LIN {X 0,Y 202.13,Z 320.552,A -85,B 0,C 180,E1 -21800.081,E2 -21800.081} C_VEL
LIN {X 0,Y 203.145,Z 321.228,A -85,B 0,C 180,E1 -21800.929,E2 -21800.929} C_VEL
LIN {X 0,Y 205.158,Z 324.532,A -85,B 0,C 180,E1 -21802.673,E2 -21802.673} C_VEL
LIN {X 0,Y 207.742,Z 326.873,A -85,B 0,C 180,E1 -21804.538,E2 -21804.538} C_VEL
LIN {X 0,Y 210.085,Z 330.227,A -85,B 0,C 180,E1 -21806.178,E2 -21806.178} C_VEL
LIN {X 0,Y 211.841,Z 332.049,A -85,B 0,C 180,E1 -21807.274,E2 -21807.274} C_VEL
LIN {X 0,Y 214.755,Z 335.87,A -85,B 0,C 180,E1 -21809.025,E2 -21809.025} C_VEL
LIN {X 0,Y 219.434,Z 342.082,A -85,B 0,C 180,E1 -21811.565,E2 -21811.565} C_VEL
LIN {X 0,Y 223.531,Z 347.82,A -85,B 0,C 180,E1 -21813.584,E2 -21813.584} C_VEL
LIN {X 0,Y 230.012,Z 357.511,A -85,B 0,C 180,E1 -21816.473,E2 -21816.473} C_VEL
LIN {X 0,Y 236.957,Z 369.03,A -85,B 0,C 180,E1 -21819.257,E2 -21819.257} C_VEL
LIN {X 0,Y 243.804,Z 381.517,A -85,B 0,C 180,E1 -21821.753,E2 -21821.753} C_VEL
LIN {X 0,Y 244.17,Z 382.3,A -85,B 0,C 180,E1 -21821.884,E2 -21821.884} C_VEL
LIN {X 0,Y 239.074,Z 460.864,A -85,B 0,C 180,E1 -21824.002,E2 -21824.002} C_VEL
LIN {X 0,Y 237.145,Z 476.486,A -85,B 0,C 180,E1 -21824.661,E2 -21824.661} C_VEL
LIN {X 0,Y 234.514,Z 492.067,A -85,B 0,C 180,E1 -21825.681,E2 -21825.681} C_VEL
LIN {X 0,Y 231.128,Z 507.018,A -85,B 0,C 180,E1 -21827.007,E2 -21827.007} C_VEL
LIN {X 0,Y 227.337,Z 520.939,A -85,B 0,C 180,E1 -21828.638,E2 -21828.638} C_VEL
LIN {X 0,Y 222.831,Z 534.369,A -85,B 0,C 180,E1 -21830.598,E2 -21830.598} C_VEL
LIN {X 0,Y 218.143,Z 546.556,A -85,B 0,C 180,E1 -21832.836,E2 -21832.836} C_VEL
LIN {X 0,Y 213.369,Z 557.823,A -85,B 0,C 180,E1 -21835.433,E2 -21835.433} C_VEL
LIN {X 0,Y 209.266,Z 566.974,A -85,B 0,C 180,E1 -21838.064,E2 -21838.064} C_VEL
LIN {X 0,Y 204.762,Z 576.14,A -85,B 0,C 180,E1 -21841.28,E2 -21841.28} C_VEL
LIN {X 0,Y 201.404,Z 582.756,A -85,B 0,C 180,E1 -21844.138,E2 -21844.138} C_VEL
LIN {X 0,Y 197.654,Z 590.063,A -85,B 0,C 180,E1 -21848.077,E2 -21848.077} C_VEL
LIN {X 0,Y 194.772,Z 595.849,A -85,B 0,C 180,E1 -21852.138,E2 -21852.138} C_VEL
LIN {X 0,Y 193.112,Z 599.272,A -85,B 0,C 180,E1 -21855.24,E2 -21855.24} C_VEL
LIN {X 0,Y 191.574,Z 602.73,A -85,B 0,C 180,E1 -21859.429,E2 -21859.429} C_VEL
LIN {X 0,Y 190.735,Z 605.008,A -85,B 0,C 180,E1 -21863.652,E2 -21863.652} C_VEL
LIN {X 0,Y 190.443,Z 606.165,A -85,B 0,C 180,E1 -21867.884,E2 -21867.884} C_VEL
LIN {X 0,Y 190.442,Z 606.176,A -85,B 0,C 180,E1 -21872.114,E2 -21872.114} C_VEL
LIN {X 0,Y 190.734,Z 605.068,A -85,B 0,C 180,E1 -21876.346,E2 -21876.346} C_VEL
LIN {X 0,Y 191.569,Z 602.836,A -85,B 0,C 180,E1 -21880.569,E2 -21880.569} C_VEL
LIN {X 0,Y 193.074,Z 599.42,A -85,B 0,C 180,E1 -21884.761,E2 -21884.761} C_VEL
LIN {X 0,Y 195.42,Z 594.732,A -85,B 0,C 180,E1 -21888.884,E2 -21888.884} C_VEL
LIN {X 0,Y 198.471,Z 588.575,A -85,B 0,C 180,E1 -21892.974,E2 -21892.974} C_VEL
LIN {X 0,Y 202.417,Z 580.99,A -85,B 0,C 180,E1 -21896.83,E2 -21896.83} C_VEL
LIN {X 0,Y 206.506,Z 572.813,A -85,B 0,C 180,E1 -21900.13,E2 -21900.13} C_VEL
LIN {X 0,Y 211.148,Z 563.18,A -85,B 0,C 180,E1 -21903.226,E2 -21903.226} C_VEL
LIN {X 0,Y 215.623,Z 552.84,A -85,B 0,C 180,E1 -21905.921,E2 -21905.921} C_VEL
LIN {X 0,Y 220.595,Z 540.782,A -85,B 0,C 180,E1 -21908.407,E2 -21908.407} C_VEL
LIN {X 0,Y 224.945,Z 528.686,A -85,B 0,C 180,E1 -21910.412,E2 -21910.412} C_VEL
LIN {X 0,Y 228.967,Z 515.537,A -85,B 0,C 180,E1 -21912.177,E2 -21912.177} C_VEL
LIN {X 0,Y 232.029,Z 503.75,A -85,B 0,C 180,E1 -21913.442,E2 -21913.442} C_VEL
LIN {X 0,Y 235.137,Z 489.584,A -85,B 0,C 180,E1 -21914.618,E2 -21914.618} C_VEL
LIN {X 0,Y 237.476,Z 475.706,A -85,B 0,C 180,E1 -21915.482,E2 -21915.482} C_VEL
LIN {X 0,Y 239.05,Z 462.425,A -85,B 0,C 180,E1 -21916.078,E2 -21916.078} C_VEL
LIN {X 0,Y 243.886,Z 390.726,A -85,B 0,C 180,E1 -21917.99,E2 -21917.99} C_VEL
LIN {X 0,Y 244.24,Z 382.256,A -85,B 0,C 180,E1 -21918.264,E2 -21918.264} C_VEL
LIN {X 0,Y 237.424,Z 369.67,A -85,B 0,C 180,E1 -21920.748,E2 -21920.748} C_VEL
LIN {X 0,Y 230.601,Z 358.379,A -85,B 0,C 180,E1 -21923.469,E2 -21923.469} C_VEL
LIN {X 0,Y 224.172,Z 348.632,A -85,B 0,C 180,E1 -21926.322,E2 -21926.322} C_VEL
LIN {X 0,Y 218.479,Z 340.65,A -85,B 0,C 180,E1 -21929.158,E2 -21929.158} C_VEL
LIN {X 0,Y 214.78,Z 335.855,A -85,B 0,C 180,E1 -21931.197,E2 -21931.197} C_VEL
LIN {X 0,Y 211.989,Z 332.222,A -85,B 0,C 180,E1 -21932.88,E2 -21932.88} C_VEL
LIN {X 0,Y 210.588,Z 330.732,A -85,B 0,C 180,E1 -21933.756,E2 -21933.756} C_VEL
LIN {X 0,Y 207.985,Z 327.314,A -85,B 0,C 180,E1 -21935.547,E2 -21935.547} C_VEL
LIN {X 0,Y 207.379,Z 326.351,A -85,B 0,C 180,E1 -21936.004,E2 -21936.004} C_VEL
LIN {X 0,Y 204.867,Z 324.176,A -85,B 0,C 180,E1 -21937.854,E2 -21937.854} C_VEL
LIN {X 0,Y 203.045,Z 321.01,A -85,B 0,C 180,E1 -21939.485,E2 -21939.485} C_VEL
LIN {X 0,Y 200.267,Z 319.057,A -85,B 0,C 180,E1 -21941.983,E2 -21941.983} C_VEL
LIN {X 0,Y 198.467,Z 316.064,A -85,B 0,C 180,E1 -21944.071,E2 -21944.071} C_VEL
LIN {X 0,Y 198.111,Z 315.123,A -85,B 0,C 180,E1 -21944.57,E2 -21944.57} C_VEL
LIN {X 0,Y 195.257,Z 313.598,A -85,B 0,C 180,E1 -21948.319,E2 -21948.319} C_VEL
LIN {X 0,Y 193.137,Z 309.963,A -85,B 0,C 180,E1 -21953.077,E2 -21953.077} C_VEL
LIN {X 0,Y 192.954,Z 309.07,A -85,B 0,C 180,E1 -21953.989,E2 -21953.989} C_VEL
LIN {X 0,Y 193.233,Z 309.035,A -85,B 0,C 180,E1 -21957.915,E2 -21957.915} C_VEL
LIN {X 0,Y 193.412,Z 309.003,A -85,B 0,C 180,E1 -21960,E2 -21960} C_VEL
LIN {X 0,Y 192.951,Z 309.06,A -85,B 0,C 180,E1 -21965.224,E2 -21965.224} C_VEL
LIN {X 0,Y 193,Z 309.378,A -85,B 0,C 180,E1 -21965.878,E2 -21965.878} C_VEL
LIN {X 0,Y 194.263,Z 312.349,A -85,B 0,C 180,E1 -21969.369,E2 -21969.369} C_VEL
LIN {X 0,Y 196.824,Z 314.644,A -85,B 0,C 180,E1 -21973.42,E2 -21973.42} C_VEL
LIN {X 0,Y 198.338,Z 315.385,A -85,B 0,C 180,E1 -21975.214,E2 -21975.214} C_VEL
LIN {X 0,Y 199.492,Z 317.921,A -85,B 0,C 180,E1 -21976.681,E2 -21976.681} C_VEL
LIN {X 0,Y 201.693,Z 320.181,A -85,B 0,C 180,E1 -21978.869,E2 -21978.869} C_VEL
LIN {X 0,Y 203.142,Z 321.115,A -85,B 0,C 180,E1 -21980.109,E2 -21980.109} C_VEL
LIN {X 0,Y 204.86,Z 324.08,A -85,B 0,C 180,E1 -21981.641,E2 -21981.641} C_VEL
LIN {X 0,Y 207.774,Z 326.812,A -85,B 0,C 180,E1 -21983.79,E2 -21983.79} C_VEL
LIN {X 0,Y 210.353,Z 330.409,A -85,B 0,C 180,E1 -21985.597,E2 -21985.597} C_VEL
LIN {X 0,Y 211.92,Z 332.086,A -85,B 0,C 180,E1 -21986.582,E2 -21986.582} C_VEL
LIN {X 0,Y 214.986,Z 336.068,A -85,B 0,C 180,E1 -21988.428,E2 -21988.428} C_VEL
LIN {X 0,Y 219.53,Z 343.033,A -85,B 0,C 180,E1 -21990.96,E2 -21990.96} C_VEL
LIN {X 0,Y 223.296,Z 349.285,A -85,B 0,C 180,E1 -21992.883,E2 -21992.883} C_VEL
LIN {X 0,Y 227.557,Z 356.613,A -85,B 0,C 180,E1 -21994.888,E2 -21994.888} C_VEL
LIN {X 0,Y 228.819,Z 359.483,A -85,B 0,C 180,E1 -21995.486,E2 -21995.486} C_VEL
LIN {X 0,Y 230.208,Z 364.449,A -85,B 0,C 180,E1 -21996.22,E2 -21996.22} C_VEL
LIN {X 0,Y 233.07,Z 378.716,A -85,B 0,C 180,E1 -21997.864,E2 -21997.864} C_VEL
LIN {X 0,Y 234.805,Z 383.494,A -85,B 0,C 180,E1 -21998.63,E2 -21998.63} C_VEL
LIN {X 0,Y 238.967,Z 393.731,A -85,B 0,C 180,E1 -22000.317,E2 -22000.317} C_VEL
LIN {X 0,Y 235.291,Z 450.409,A -85,B 0,C 180,E1 -22001.853,E2 -22001.853} C_VEL
LIN {X 0,Y 233.436,Z 475.234,A -85,B 0,C 180,E1 -22002.552,E2 -22002.552} C_VEL
LIN {X 0,Y 231.252,Z 490.946,A -85,B 0,C 180,E1 -22003.245,E2 -22003.245} C_VEL
LIN {X 0,Y 228.371,Z 505.434,A -85,B 0,C 180,E1 -22004.158,E2 -22004.158} C_VEL
LIN {X 0,Y 224.872,Z 519.174,A -85,B 0,C 180,E1 -22005.317,E2 -22005.317} C_VEL
LIN {X 0,Y 220.787,Z 532.642,A -85,B 0,C 180,E1 -22006.814,E2 -22006.814} C_VEL
LIN {X 0,Y 216.512,Z 544.93,A -85,B 0,C 180,E1 -22008.562,E2 -22008.562} C_VEL
LIN {X 0,Y 211.366,Z 557.724,A -85,B 0,C 180,E1 -22010.821,E2 -22010.821} C_VEL
LIN {X 0,Y 206.254,Z 569.229,A -85,B 0,C 180,E1 -22013.395,E2 -22013.395} C_VEL
LIN {X 0,Y 201.601,Z 578.92,A -85,B 0,C 180,E1 -22016.099,E2 -22016.099} C_VEL
LIN {X 0,Y 196.862,Z 588.577,A -85,B 0,C 180,E1 -22019.481,E2 -22019.481} C_VEL
LIN {X 0,Y 192.876,Z 596.405,A -85,B 0,C 180,E1 -22022.906,E2 -22022.906} C_VEL
LIN {X 0,Y 189.093,Z 603.84,A -85,B 0,C 180,E1 -22027.031,E2 -22027.031} C_VEL
LIN {X 0,Y 186.295,Z 609.751,A -85,B 0,C 180,E1 -22031.298,E2 -22031.298} C_VEL
LIN {X 0,Y 184.799,Z 613.274,A -85,B 0,C 180,E1 -22034.562,E2 -22034.562} C_VEL
LIN {X 0,Y 183.53,Z 616.842,A -85,B 0,C 180,E1 -22038.963,E2 -22038.963} C_VEL
LIN {X 0,Y 183.109,Z 619.202,A -85,B 0,C 180,E1 -22043.389,E2 -22043.389} C_VEL
LIN {X 0,Y 183.13,Z 620.394,A -85,B 0,C 180,E1 -22047.802,E2 -22047.802} C_VEL
LIN {X 0,Y 183.283,Z 620.556,A -85,B 0,C 180,E1 -22050.001,E2 -22050.001} C_VEL
LIN {X 0,Y 183.114,Z 619.928,A -85,B 0,C 180,E1 -22054.403,E2 -22054.403} C_VEL
LIN {X 0,Y 183.241,Z 618.133,A -85,B 0,C 180,E1 -22058.826,E2 -22058.826} C_VEL
LIN {X 0,Y 184.022,Z 615.159,A -85,B 0,C 180,E1 -22063.248,E2 -22063.248} C_VEL
LIN {X 0,Y 185.723,Z 610.945,A -85,B 0,C 180,E1 -22067.623,E2 -22067.623} C_VEL
LIN {X 0,Y 188.26,Z 605.378,A -85,B 0,C 180,E1 -22071.921,E2 -22071.921} C_VEL
LIN {X 0,Y 191.758,Z 598.315,A -85,B 0,C 180,E1 -22076.093,E2 -22076.093} C_VEL
LIN {X 0,Y 195.731,Z 590.779,A -85,B 0,C 180,E1 -22079.586,E2 -22079.586} C_VEL
LIN {X 0,Y 200.221,Z 581.697,A -85,B 0,C 180,E1 -22082.962,E2 -22082.962} C_VEL
LIN {X 0,Y 205.441,Z 570.793,A -85,B 0,C 180,E1 -22086.166,E2 -22086.166} C_VEL
LIN {X 0,Y 210.422,Z 559.576,A -85,B 0,C 180,E1 -22088.775,E2 -22088.775} C_VEL
LIN {X 0,Y 215.782,Z 546.661,A -85,B 0,C 180,E1 -22091.121,E2 -22091.121} C_VEL
LIN {X 0,Y 220.293,Z 533.792,A -85,B 0,C 180,E1 -22092.996,E2 -22092.996} C_VEL
LIN {X 0,Y 224.342,Z 520.525,A -85,B 0,C 180,E1 -22094.504,E2 -22094.504} C_VEL
LIN {X 0,Y 227.806,Z 507.143,A -85,B 0,C 180,E1 -22095.673,E2 -22095.673} C_VEL
LIN {X 0,Y 230.83,Z 492.493,A -85,B 0,C 180,E1 -22096.63,E2 -22096.63} C_VEL
LIN {X 0,Y 232.989,Z 477.524,A -85,B 0,C 180,E1 -22097.331,E2 -22097.331} C_VEL
LIN {X 0,Y 234.684,Z 457.569,A -85,B 0,C 180,E1 -22097.913,E2 -22097.913} C_VEL
LIN {X 0,Y 238.816,Z 393.594,A -85,B 0,C 180,E1 -22099.652,E2 -22099.652} C_VEL
LIN {X 0,Y 233.193,Z 380.016,A -85,B 0,C 180,E1 -22101.945,E2 -22101.945} C_VEL
LIN {X 0,Y 227.753,Z 368.646,A -85,B 0,C 180,E1 -22104.303,E2 -22104.303} C_VEL
LIN {X 0,Y 221.581,Z 356.972,A -85,B 0,C 180,E1 -22107.236,E2 -22107.236} C_VEL
LIN {X 0,Y 215.921,Z 347.368,A -85,B 0,C 180,E1 -22110.24,E2 -22110.24} C_VEL
LIN {X 0,Y 212.629,Z 342.242,A -85,B 0,C 180,E1 -22112.169,E2 -22112.169} C_VEL
LIN {X 0,Y 208.968,Z 337.475,A -85,B 0,C 180,E1 -22114.475,E2 -22114.475} C_VEL
LIN {X 0,Y 206.188,Z 333.97,A -85,B 0,C 180,E1 -22116.414,E2 -22116.414} C_VEL
LIN {X 0,Y 205.461,Z 332.88,A -85,B 0,C 180,E1 -22116.971,E2 -22116.971} C_VEL
LIN {X 0,Y 202.738,Z 330.139,A -85,B 0,C 180,E1 -22119.088,E2 -22119.088} C_VEL
LIN {X 0,Y 201.362,Z 327.685,A -85,B 0,C 180,E1 -22120.371,E2 -22120.371} C_VEL
LIN {X 0,Y 198.647,Z 325.483,A -85,B 0,C 180,E1 -22122.918,E2 -22122.918} C_VEL
LIN {X 0,Y 196.975,Z 322.515,A -85,B 0,C 180,E1 -22124.942,E2 -22124.942} C_VEL
LIN {X 0,Y 196.531,Z 321.931,A -85,B 0,C 180,E1 -22125.504,E2 -22125.504} C_VEL
LIN {X 0,Y 193.771,Z 320.059,A -85,B 0,C 180,E1 -22129.354,E2 -22129.354} C_VEL
LIN {X 0,Y 192.084,Z 316.757,A -85,B 0,C 180,E1 -22133.303,E2 -22133.303} C_VEL
LIN {X 0,Y 191.818,Z 316.073,A -85,B 0,C 180,E1 -22134.217,E2 -22134.217} C_VEL
LIN {X 0,Y 190.8,Z 315.614,A -85,B 0,C 180,E1 -22140,E2 -22140} C_VEL
LIN {X 0,Y 192.014,Z 316.301,A -85,B 0,C 180,E1 -22146.964,E2 -22146.964} C_VEL
LIN {X 0,Y 193.236,Z 319.399,A -85,B 0,C 180,E1 -22150.234,E2 -22150.234} C_VEL
LIN {X 0,Y 195.466,Z 321.51,A -85,B 0,C 180,E1 -22153.781,E2 -22153.781} C_VEL
LIN {X 0,Y 196.819,Z 322.191,A -85,B 0,C 180,E1 -22155.428,E2 -22155.428} C_VEL
LIN {X 0,Y 198.612,Z 325.558,A -85,B 0,C 180,E1 -22157.64,E2 -22157.64} C_VEL
LIN {X 0,Y 201.56,Z 328.097,A -85,B 0,C 180,E1 -22160.407,E2 -22160.407} C_VEL
LIN {X 0,Y 203.71,Z 331.392,A -85,B 0,C 180,E1 -22162.303,E2 -22162.303} C_VEL
LIN {X 0,Y 205.811,Z 333.361,A -85,B 0,C 180,E1 -22163.876,E2 -22163.876} C_VEL
LIN {X 0,Y 208.392,Z 336.945,A -85,B 0,C 180,E1 -22165.735,E2 -22165.735} C_VEL
LIN {X 0,Y 209.758,Z 338.468,A -85,B 0,C 180,E1 -22166.624,E2 -22166.624} C_VEL
LIN {X 0,Y 212.93,Z 342.541,A -85,B 0,C 180,E1 -22168.584,E2 -22168.584} C_VEL
LIN {X 0,Y 219.429,Z 351.601,A -85,B 0,C 180,E1 -22172.146,E2 -22172.146} C_VEL
LIN {X 0,Y 226.743,Z 362.814,A -85,B 0,C 180,E1 -22175.613,E2 -22175.613} C_VEL
LIN {X 0,Y 233.269,Z 373.858,A -85,B 0,C 180,E1 -22178.36,E2 -22178.36} C_VEL
LIN {X 0,Y 239.321,Z 385.095,A -85,B 0,C 180,E1 -22180.686,E2 -22180.686} C_VEL
LIN {X 0,Y 234.217,Z 461.153,A -85,B 0,C 180,E1 -22182.757,E2 -22182.757} C_VEL
LIN {X 0,Y 232.232,Z 476.767,A -85,B 0,C 180,E1 -22183.421,E2 -22183.421} C_VEL
LIN {X 0,Y 229.486,Z 492.346,A -85,B 0,C 180,E1 -22184.442,E2 -22184.442} C_VEL
LIN {X 0,Y 226.006,Z 507.293,A -85,B 0,C 180,E1 -22185.785,E2 -22185.785} C_VEL
LIN {X 0,Y 222.066,Z 521.214,A -85,B 0,C 180,E1 -22187.429,E2 -22187.429} C_VEL
LIN {X 0,Y 217.393,Z 534.643,A -85,B 0,C 180,E1 -22189.411,E2 -22189.411} C_VEL
LIN {X 0,Y 212.518,Z 546.83,A -85,B 0,C 180,E1 -22191.678,E2 -22191.678} C_VEL
LIN {X 0,Y 207.556,Z 558.097,A -85,B 0,C 180,E1 -22194.32,E2 -22194.32} C_VEL
LIN {X 0,Y 202.524,Z 568.691,A -85,B 0,C 180,E1 -22197.459,E2 -22197.459} C_VEL
LIN {X 0,Y 197.926,Z 577.626,A -85,B 0,C 180,E1 -22200.774,E2 -22200.774} C_VEL
LIN {X 0,Y 193.952,Z 585.023,A -85,B 0,C 180,E1 -22204.224,E2 -22204.224} C_VEL
LIN {X 0,Y 190.243,Z 591.928,A -85,B 0,C 180,E1 -22208.319,E2 -22208.319} C_VEL
LIN {X 0,Y 187.299,Z 597.347,A -85,B 0,C 180,E1 -22212.53,E2 -22212.53} C_VEL
LIN {X 0,Y 185.313,Z 601.425,A -85,B 0,C 180,E1 -22216.846,E2 -22216.846} C_VEL
LIN {X 0,Y 184.05,Z 604.284,A -85,B 0,C 180,E1 -22221.213,E2 -22221.213} C_VEL
LIN {X 0,Y 183.449,Z 605.995,A -85,B 0,C 180,E1 -22225.605,E2 -22225.605} C_VEL
LIN {X 0,Y 183.336,Z 606.589,A -85,B 0,C 180,E1 -22229.999,E2 -22229.999} C_VEL
LIN {X 0,Y 183.449,Z 606.031,A -85,B 0,C 180,E1 -22234.393,E2 -22234.393} C_VEL
LIN {X 0,Y 184.048,Z 604.366,A -85,B 0,C 180,E1 -22238.785,E2 -22238.785} C_VEL
LIN {X 0,Y 185.295,Z 601.551,A -85,B 0,C 180,E1 -22243.153,E2 -22243.153} C_VEL
LIN {X 0,Y 187.249,Z 597.515,A -85,B 0,C 180,E1 -22247.472,E2 -22247.472} C_VEL
LIN {X 0,Y 190.147,Z 592.15,A -85,B 0,C 180,E1 -22251.69,E2 -22251.69} C_VEL
LIN {X 0,Y 193.855,Z 585.308,A -85,B 0,C 180,E1 -22255.787,E2 -22255.787} C_VEL
LIN {X 0,Y 198.454,Z 576.755,A -85,B 0,C 180,E1 -22259.721,E2 -22259.721} C_VEL
LIN {X 0,Y 203.204,Z 567.65,A -85,B 0,C 180,E1 -22263.005,E2 -22263.005} C_VEL
LIN {X 0,Y 207.421,Z 558.546,A -85,B 0,C 180,E1 -22265.705,E2 -22265.705} C_VEL
LIN {X 0,Y 212.458,Z 547.353,A -85,B 0,C 180,E1 -22268.333,E2 -22268.333} C_VEL
LIN {X 0,Y 217.255,Z 535.27,A -85,B 0,C 180,E1 -22270.618,E2 -22270.618} C_VEL
LIN {X 0,Y 221.912,Z 521.99,A -85,B 0,C 180,E1 -22272.605,E2 -22272.605} C_VEL
LIN {X 0,Y 225.604,Z 509.172,A -85,B 0,C 180,E1 -22274.151,E2 -22274.151} C_VEL
LIN {X 0,Y 229.127,Z 494.706,A -85,B 0,C 180,E1 -22275.49,E2 -22275.49} C_VEL
LIN {X 0,Y 231.901,Z 480.025,A -85,B 0,C 180,E1 -22276.505,E2 -22276.505} C_VEL
LIN {X 0,Y 233.94,Z 464.955,A -85,B 0,C 180,E1 -22277.234,E2 -22277.234} C_VEL
LIN {X 0,Y 235.343,Z 448.353,A -85,B 0,C 180,E1 -22277.734,E2 -22277.734} C_VEL
LIN {X 0,Y 239.471,Z 385.303,A -85,B 0,C 180,E1 -22279.433,E2 -22279.433} C_VEL
LIN {X 0,Y 232.955,Z 373.112,A -85,B 0,C 180,E1 -22281.956,E2 -22281.956} C_VEL
LIN {X 0,Y 226.004,Z 361.512,A -85,B 0,C 180,E1 -22284.917,E2 -22284.917} C_VEL
LIN {X 0,Y 218.751,Z 350.547,A -85,B 0,C 180,E1 -22288.42,E2 -22288.42} C_VEL
LIN {X 0,Y 214.628,Z 345.033,A -85,B 0,C 180,E1 -22290.647,E2 -22290.647} C_VEL
LIN {X 0,Y 212.452,Z 342.032,A -85,B 0,C 180,E1 -22291.931,E2 -22291.931} C_VEL
LIN {X 0,Y 209.066,Z 337.592,A -85,B 0,C 180,E1 -22294.086,E2 -22294.086} C_VEL
LIN {X 0,Y 206.32,Z 334.216,A -85,B 0,C 180,E1 -22296.006,E2 -22296.006} C_VEL
LIN {X 0,Y 205.42,Z 332.907,A -85,B 0,C 180,E1 -22296.697,E2 -22296.697} C_VEL
LIN {X 0,Y 202.711,Z 330.117,A -85,B 0,C 180,E1 -22298.838,E2 -22298.838} C_VEL
LIN {X 0,Y 201.303,Z 327.686,A -85,B 0,C 180,E1 -22300.165,E2 -22300.165} C_VEL
LIN {X 0,Y 198.685,Z 325.586,A -85,B 0,C 180,E1 -22302.661,E2 -22302.661} C_VEL
LIN {X 0,Y 196.905,Z 322.419,A -85,B 0,C 180,E1 -22304.87,E2 -22304.87} C_VEL
LIN {X 0,Y 196.412,Z 321.915,A -85,B 0,C 180,E1 -22305.494,E2 -22305.494} C_VEL
LIN {X 0,Y 193.762,Z 320.069,A -85,B 0,C 180,E1 -22309.367,E2 -22309.367} C_VEL
LIN {X 0,Y 191.99,Z 316.273,A -85,B 0,C 180,E1 -22314.09,E2 -22314.09} C_VEL
LIN {X 0,Y 191.122,Z 315.724,A -85,B 0,C 180,E1 -22320,E2 -22320} C_VEL
LIN {X 0,Y 191.984,Z 316.219,A -85,B 0,C 180,E1 -22325.382,E2 -22325.382} C_VEL
LIN {X 0,Y 193.28,Z 319.362,A -85,B 0,C 180,E1 -22329.175,E2 -22329.175} C_VEL
LIN {X 0,Y 195.593,Z 321.528,A -85,B 0,C 180,E1 -22332.978,E2 -22332.978} C_VEL
LIN {X 0,Y 196.899,Z 322.186,A -85,B 0,C 180,E1 -22334.601,E2 -22334.601} C_VEL
LIN {X 0,Y 198.354,Z 325.041,A -85,B 0,C 180,E1 -22336.466,E2 -22336.466} C_VEL
LIN {X 0,Y 200.658,Z 327.228,A -85,B 0,C 180,E1 -22338.771,E2 -22338.771} C_VEL
LIN {X 0,Y 201.545,Z 327.96,A -85,B 0,C 180,E1 -22339.564,E2 -22339.564} C_VEL
LIN {X 0,Y 203.71,Z 331.292,A -85,B 0,C 180,E1 -22341.504,E2 -22341.504} C_VEL
LIN {X 0,Y 205.872,Z 333.311,A -85,B 0,C 180,E1 -22343.14,E2 -22343.14} C_VEL
LIN {X 0,Y 208.65,Z 337.112,A -85,B 0,C 180,E1 -22345.146,E2 -22345.146} C_VEL
LIN {X 0,Y 210.023,Z 338.805,A -85,B 0,C 180,E1 -22346.053,E2 -22346.053} C_VEL
LIN {X 0,Y 213.649,Z 343.667,A -85,B 0,C 180,E1 -22348.294,E2 -22348.294} C_VEL
LIN {X 0,Y 217.814,Z 350.47,A -85,B 0,C 180,E1 -22350.677,E2 -22350.677} C_VEL
LIN {X 0,Y 222.059,Z 357.794,A -85,B 0,C 180,E1 -22352.887,E2 -22352.887} C_VEL
LIN {X 0,Y 227.28,Z 367.659,A -85,B 0,C 180,E1 -22355.38,E2 -22355.38} C_VEL
LIN {X 0,Y 232.625,Z 378.602,A -85,B 0,C 180,E1 -22357.719,E2 -22357.719} C_VEL
LIN {X 0,Y 234.805,Z 383.494,A -85,B 0,C 180,E1 -22358.63,E2 -22358.63} C_VEL
LIN {X 0,Y 235.574,Z 386.228,A -85,B 0,C 180,E1 -22358.99,E2 -22358.99} C_VEL
LIN {X 0,Y 235.666,Z 390.703,A -85,B 0,C 180,E1 -22359.228,E2 -22359.228} C_VEL
LIN {X 0,Y 233.874,Z 403.174,A -85,B 0,C 180,E1 -22359.285,E2 -22359.285} C_VEL
LIN {X 0,Y 233.774,Z 404.58,A -85,B 0,C 180,E1 -22359.322,E2 -22359.322} C_VEL
LIN {X 0,Y 228.83,Z 473.789,A -85,B 0,C 180,E1 -22361.197,E2 -22361.197} C_VEL
LIN {X 0,Y 226.566,Z 489.92,A -85,B 0,C 180,E1 -22361.887,E2 -22361.887} C_VEL
LIN {X 0,Y 223.458,Z 505.169,A -85,B 0,C 180,E1 -22362.846,E2 -22362.846} C_VEL
LIN {X 0,Y 219.862,Z 518.908,A -85,B 0,C 180,E1 -22364.011,E2 -22364.011} C_VEL
LIN {X 0,Y 215.646,Z 532.376,A -85,B 0,C 180,E1 -22365.518,E2 -22365.518} C_VEL
LIN {X 0,Y 211.045,Z 545.121,A -85,B 0,C 180,E1 -22367.353,E2 -22367.353} C_VEL
LIN {X 0,Y 205.879,Z 557.456,A -85,B 0,C 180,E1 -22369.565,E2 -22369.565} C_VEL
LIN {X 0,Y 200.564,Z 568.959,A -85,B 0,C 180,E1 -22372.178,E2 -22372.178} C_VEL
LIN {X 0,Y 195.692,Z 578.649,A -85,B 0,C 180,E1 -22374.928,E2 -22374.928} C_VEL
LIN {X 0,Y 190.911,Z 587.945,A -85,B 0,C 180,E1 -22378.242,E2 -22378.242} C_VEL
LIN {X 0,Y 186.513,Z 596.133,A -85,B 0,C 180,E1 -22381.901,E2 -22381.901} C_VEL
LIN {X 0,Y 182.497,Z 603.567,A -85,B 0,C 180,E1 -22386.15,E2 -22386.15} C_VEL
LIN {X 0,Y 179.513,Z 609.478,A -85,B 0,C 180,E1 -22390.564,E2 -22390.564} C_VEL
LIN {X 0,Y 177.901,Z 613.002,A -85,B 0,C 180,E1 -22393.948,E2 -22393.948} C_VEL
LIN {X 0,Y 176.508,Z 616.57,A -85,B 0,C 180,E1 -22398.518,E2 -22398.518} C_VEL
LIN {X 0,Y 176.013,Z 618.93,A -85,B 0,C 180,E1 -22403.121,E2 -22403.121} C_VEL
LIN {X 0,Y 176.015,Z 619.921,A -85,B 0,C 180,E1 -22406.569,E2 -22406.569} C_VEL
LIN {X 0,Y 176.185,Z 620.285,A -85,B 0,C 180,E1 -22410.001,E2 -22410.001} C_VEL
LIN {X 0,Y 176.019,Z 619.657,A -85,B 0,C 180,E1 -22414.581,E2 -22414.581} C_VEL
LIN {X 0,Y 176.19,Z 617.861,A -85,B 0,C 180,E1 -22419.182,E2 -22419.182} C_VEL
LIN {X 0,Y 177.051,Z 614.885,A -85,B 0,C 180,E1 -22423.78,E2 -22423.78} C_VEL
LIN {X 0,Y 178.906,Z 610.671,A -85,B 0,C 180,E1 -22428.318,E2 -22428.318} C_VEL
LIN {X 0,Y 181.61,Z 605.103,A -85,B 0,C 180,E1 -22432.768,E2 -22432.768} C_VEL
LIN {X 0,Y 185.338,Z 598.04,A -85,B 0,C 180,E1 -22437.069,E2 -22437.069} C_VEL
LIN {X 0,Y 189.49,Z 590.503,A -85,B 0,C 180,E1 -22440.663,E2 -22440.663} C_VEL
LIN {X 0,Y 194.241,Z 581.421,A -85,B 0,C 180,E1 -22444.114,E2 -22444.114} C_VEL
LIN {X 0,Y 199.712,Z 570.518,A -85,B 0,C 180,E1 -22447.377,E2 -22447.377} C_VEL
LIN {X 0,Y 204.919,Z 559.302,A -85,B 0,C 180,E1 -22450.022,E2 -22450.022} C_VEL
LIN {X 0,Y 210.373,Z 546.589,A -85,B 0,C 180,E1 -22452.366,E2 -22452.366} C_VEL
LIN {X 0,Y 215.14,Z 533.516,A -85,B 0,C 180,E1 -22454.289,E2 -22454.289} C_VEL
LIN {X 0,Y 219.305,Z 520.248,A -85,B 0,C 180,E1 -22455.813,E2 -22455.813} C_VEL
LIN {X 0,Y 222.878,Z 506.864,A -85,B 0,C 180,E1 -22456.986,E2 -22456.986} C_VEL
LIN {X 0,Y 226.014,Z 492.213,A -85,B 0,C 180,E1 -22457.938,E2 -22457.938} C_VEL
LIN {X 0,Y 228.247,Z 477.24,A -85,B 0,C 180,E1 -22458.638,E2 -22458.638} C_VEL
LIN {X 0,Y 229.989,Z 457.277,A -85,B 0,C 180,E1 -22459.225,E2 -22459.225} C_VEL
LIN {X 0,Y 234.146,Z 396.149,A -85,B 0,C 180,E1 -22460.881,E2 -22460.881} C_VEL
LIN {X 0,Y 228.792,Z 383.138,A -85,B 0,C 180,E1 -22463.201,E2 -22463.201} C_VEL
LIN {X 0,Y 223.37,Z 371.735,A -85,B 0,C 180,E1 -22465.709,E2 -22465.709} C_VEL
LIN {X 0,Y 218.249,Z 361.872,A -85,B 0,C 180,E1 -22468.306,E2 -22468.306} C_VEL
LIN {X 0,Y 213.174,Z 352.979,A -85,B 0,C 180,E1 -22471.159,E2 -22471.159} C_VEL
LIN {X 0,Y 210.264,Z 348.333,A -85,B 0,C 180,E1 -22472.952,E2 -22472.952} C_VEL
LIN {X 0,Y 206.729,Z 343.627,A -85,B 0,C 180,E1 -22475.289,E2 -22475.289} C_VEL
LIN {X 0,Y 203.919,Z 339.743,A -85,B 0,C 180,E1 -22477.381,E2 -22477.381} C_VEL
LIN {X 0,Y 200.753,Z 336.231,A -85,B 0,C 180,E1 -22479.976,E2 -22479.976} C_VEL
LIN {X 0,Y 199.706,Z 334.347,A -85,B 0,C 180,E1 -22481.003,E2 -22481.003} C_VEL
LIN {X 0,Y 197.123,Z 332.045,A -85,B 0,C 180,E1 -22483.561,E2 -22483.561} C_VEL
LIN {X 0,Y 195.266,Z 328.846,A -85,B 0,C 180,E1 -22485.94,E2 -22485.94} C_VEL
LIN {X 0,Y 192.666,Z 326.943,A -85,B 0,C 180,E1 -22489.735,E2 -22489.735} C_VEL
LIN {X 0,Y 191.011,Z 323.457,A -85,B 0,C 180,E1 -22493.928,E2 -22493.928} C_VEL
LIN {X 0,Y 190.784,Z 323.072,A -85,B 0,C 180,E1 -22494.716,E2 -22494.716} C_VEL
LIN {X 0,Y 190.016,Z 322.767,A -85,B 0,C 180,E1 -22502.12,E2 -22502.12} C_VEL
LIN {X 0,Y 191.031,Z 323.349,A -85,B 0,C 180,E1 -22506.671,E2 -22506.671} C_VEL
LIN {X 0,Y 192.218,Z 326.384,A -85,B 0,C 180,E1 -22509.982,E2 -22509.982} C_VEL
LIN {X 0,Y 194.429,Z 328.503,A -85,B 0,C 180,E1 -22513.589,E2 -22513.589} C_VEL
LIN {X 0,Y 195.512,Z 329.22,A -85,B 0,C 180,E1 -22514.973,E2 -22514.973} C_VEL
LIN {X 0,Y 197.475,Z 332.617,A -85,B 0,C 180,E1 -22517.425,E2 -22517.425} C_VEL
LIN {X 0,Y 199.963,Z 334.84,A -85,B 0,C 180,E1 -22519.84,E2 -22519.84} C_VEL
LIN {X 0,Y 202.275,Z 338.26,A -85,B 0,C 180,E1 -22521.932,E2 -22521.932} C_VEL
LIN {X 0,Y 204.035,Z 340.063,A -85,B 0,C 180,E1 -22523.305,E2 -22523.305} C_VEL
LIN {X 0,Y 206.839,Z 343.771,A -85,B 0,C 180,E1 -22525.369,E2 -22525.369} C_VEL
LIN {X 0,Y 208.358,Z 345.911,A -85,B 0,C 180,E1 -22526.412,E2 -22526.412} C_VEL
LIN {X 0,Y 211.418,Z 349.959,A -85,B 0,C 180,E1 -22528.343,E2 -22528.343} C_VEL
LIN {X 0,Y 215.3,Z 355.452,A -85,B 0,C 180,E1 -22530.582,E2 -22530.582} C_VEL
LIN {X 0,Y 220.296,Z 363.001,A -85,B 0,C 180,E1 -22533.184,E2 -22533.184} C_VEL
LIN {X 0,Y 226.01,Z 372.328,A -85,B 0,C 180,E1 -22535.862,E2 -22535.862} C_VEL
LIN {X 0,Y 232.346,Z 383.678,A -85,B 0,C 180,E1 -22538.551,E2 -22538.551} C_VEL
LIN {X 0,Y 234.617,Z 388.371,A -85,B 0,C 180,E1 -22539.472,E2 -22539.472} C_VEL
LIN {X 0,Y 229.425,Z 462.021,A -85,B 0,C 180,E1 -22541.479,E2 -22541.479} C_VEL
LIN {X 0,Y 227.272,Z 477.92,A -85,B 0,C 180,E1 -22542.166,E2 -22542.166} C_VEL
LIN {X 0,Y 224.589,Z 492.624,A -85,B 0,C 180,E1 -22543.153,E2 -22543.153} C_VEL
LIN {X 0,Y 220.987,Z 507.564,A -85,B 0,C 180,E1 -22544.504,E2 -22544.504} C_VEL
LIN {X 0,Y 216.901,Z 521.488,A -85,B 0,C 180,E1 -22546.163,E2 -22546.163} C_VEL
LIN {X 0,Y 212.062,Z 534.917,A -85,B 0,C 180,E1 -22548.165,E2 -22548.165} C_VEL
LIN {X 0,Y 206.999,Z 547.104,A -85,B 0,C 180,E1 -22550.46,E2 -22550.46} C_VEL
LIN {X 0,Y 201.826,Z 558.37,A -85,B 0,C 180,E1 -22553.143,E2 -22553.143} C_VEL
LIN {X 0,Y 196.578,Z 568.964,A -85,B 0,C 180,E1 -22556.346,E2 -22556.346} C_VEL
LIN {X 0,Y 191.747,Z 577.899,A -85,B 0,C 180,E1 -22559.736,E2 -22559.736} C_VEL
LIN {X 0,Y 187.547,Z 585.297,A -85,B 0,C 180,E1 -22563.276,E2 -22563.276} C_VEL
LIN {X 0,Y 183.613,Z 592.202,A -85,B 0,C 180,E1 -22567.494,E2 -22567.494} C_VEL
LIN {X 0,Y 180.517,Z 597.62,A -85,B 0,C 180,E1 -22571.851,E2 -22571.851} C_VEL
LIN {X 0,Y 178.385,Z 601.697,A -85,B 0,C 180,E1 -22576.325,E2 -22576.325} C_VEL
LIN {X 0,Y 177.036,Z 604.555,A -85,B 0,C 180,E1 -22580.862,E2 -22580.862} C_VEL
LIN {X 0,Y 176.391,Z 606.265,A -85,B 0,C 180,E1 -22585.428,E2 -22585.428} C_VEL
LIN {X 0,Y 176.241,Z 606.859,A -85,B 0,C 180,E1 -22589.999,E2 -22589.999} C_VEL
LIN {X 0,Y 176.39,Z 606.3,A -85,B 0,C 180,E1 -22594.569,E2 -22594.569} C_VEL
LIN {X 0,Y 177.034,Z 604.636,A -85,B 0,C 180,E1 -22599.136,E2 -22599.136} C_VEL
LIN {X 0,Y 178.364,Z 601.821,A -85,B 0,C 180,E1 -22603.674,E2 -22603.674} C_VEL
LIN {X 0,Y 180.467,Z 597.785,A -85,B 0,C 180,E1 -22608.151,E2 -22608.151} C_VEL
LIN {X 0,Y 183.523,Z 592.421,A -85,B 0,C 180,E1 -22612.515,E2 -22612.515} C_VEL
LIN {X 0,Y 187.46,Z 585.578,A -85,B 0,C 180,E1 -22616.735,E2 -22616.735} C_VEL
LIN {X 0,Y 192.316,Z 577.023,A -85,B 0,C 180,E1 -22620.77,E2 -22620.77} C_VEL
LIN {X 0,Y 197.28,Z 567.918,A -85,B 0,C 180,E1 -22624.13,E2 -22624.13} C_VEL
LIN {X 0,Y 201.77,Z 558.651,A -85,B 0,C 180,E1 -22626.93,E2 -22626.93} C_VEL
LIN {X 0,Y 207.381,Z 546.63,A -85,B 0,C 180,E1 -22629.765,E2 -22629.765} C_VEL
LIN {X 0,Y 212.373,Z 534.353,A -85,B 0,C 180,E1 -22632.076,E2 -22632.076} C_VEL
LIN {X 0,Y 217.218,Z 520.789,A -85,B 0,C 180,E1 -22634.076,E2 -22634.076} C_VEL
LIN {X 0,Y 221.324,Z 506.628,A -85,B 0,C 180,E1 -22635.739,E2 -22635.739} C_VEL
LIN {X 0,Y 224.709,Z 492.692,A -85,B 0,C 180,E1 -22636.976,E2 -22636.976} C_VEL
LIN {X 0,Y 227.636,Z 477.135,A -85,B 0,C 180,E1 -22637.978,E2 -22637.978} C_VEL
LIN {X 0,Y 229.457,Z 462.934,A -85,B 0,C 180,E1 -22638.625,E2 -22638.625} C_VEL
LIN {X 0,Y 234.682,Z 390.552,A -85,B 0,C 180,E1 -22640.581,E2 -22640.581} C_VEL
LIN {X 0,Y 234.684,Z 388.116,A -85,B 0,C 180,E1 -22640.696,E2 -22640.696} C_VEL
LIN {X 0,Y 228.44,Z 376.366,A -85,B 0,C 180,E1 -22643.272,E2 -22643.272} C_VEL
LIN {X 0,Y 222.173,Z 365.842,A -85,B 0,C 180,E1 -22646.115,E2 -22646.115} C_VEL
LIN {X 0,Y 216.139,Z 356.486,A -85,B 0,C 180,E1 -22649.194,E2 -22649.194} C_VEL
LIN {X 0,Y 212.317,Z 351.207,A -85,B 0,C 180,E1 -22651.354,E2 -22651.354} C_VEL
LIN {X 0,Y 210.106,Z 348.096,A -85,B 0,C 180,E1 -22652.718,E2 -22652.718} C_VEL
LIN {X 0,Y 206.9,Z 343.818,A -85,B 0,C 180,E1 -22654.857,E2 -22654.857} C_VEL
LIN {X 0,Y 204.097,Z 340.079,A -85,B 0,C 180,E1 -22656.94,E2 -22656.94} C_VEL
LIN {X 0,Y 200.699,Z 336.141,A -85,B 0,C 180,E1 -22659.769,E2 -22659.769} C_VEL
LIN {X 0,Y 199.727,Z 334.405,A -85,B 0,C 180,E1 -22660.738,E2 -22660.738} C_VEL
LIN {X 0,Y 197.069,Z 332.037,A -85,B 0,C 180,E1 -22663.423,E2 -22663.423} C_VEL
LIN {X 0,Y 195.365,Z 328.911,A -85,B 0,C 180,E1 -22665.681,E2 -22665.681} C_VEL
LIN {X 0,Y 192.687,Z 326.986,A -85,B 0,C 180,E1 -22669.716,E2 -22669.716} C_VEL
LIN {X 0,Y 190.953,Z 323.081,A -85,B 0,C 180,E1 -22674.72,E2 -22674.72} C_VEL
LIN {X 0,Y 190.4,Z 322.899,A -85,B 0,C 180,E1 -22682.115,E2 -22682.115} C_VEL
LIN {X 0,Y 191.03,Z 323.335,A -85,B 0,C 180,E1 -22685.145,E2 -22685.145} C_VEL
LIN {X 0,Y 192.808,Z 327.079,A -85,B 0,C 180,E1 -22690.013,E2 -22690.013} C_VEL
LIN {X 0,Y 195.617,Z 329.235,A -85,B 0,C 180,E1 -22694.167,E2 -22694.167} C_VEL
LIN {X 0,Y 197.262,Z 332.171,A -85,B 0,C 180,E1 -22696.294,E2 -22696.294} C_VEL
LIN {X 0,Y 199.938,Z 334.668,A -85,B 0,C 180,E1 -22698.974,E2 -22698.974} C_VEL
LIN {X 0,Y 202.279,Z 338.149,A -85,B 0,C 180,E1 -22701.129,E2 -22701.129} C_VEL
LIN {X 0,Y 204.135,Z 339.996,A -85,B 0,C 180,E1 -22702.587,E2 -22702.587} C_VEL
LIN {X 0,Y 206.952,Z 343.811,A -85,B 0,C 180,E1 -22704.683,E2 -22704.683} C_VEL
LIN {X 0,Y 211.227,Z 349.668,A -85,B 0,C 180,E1 -22707.494,E2 -22707.494} C_VEL
LIN {X 0,Y 215.842,Z 357.452,A -85,B 0,C 180,E1 -22710.243,E2 -22710.243} C_VEL
LIN {X 0,Y 221.713,Z 368.206,A -85,B 0,C 180,E1 -22713.351,E2 -22713.351} C_VEL
LIN {X 0,Y 227.657,Z 380.507,A -85,B 0,C 180,E1 -22716.186,E2 -22716.186} C_VEL
LIN {X 0,Y 232.257,Z 391.132,A -85,B 0,C 180,E1 -22718.216,E2 -22718.216} C_VEL
LIN {X 0,Y 234.233,Z 396.08,A -85,B 0,C 180,E1 -22719.056,E2 -22719.056} C_VEL
LIN {X 0,Y 233.774,Z 404.58,A -85,B 0,C 180,E1 -22719.322,E2 -22719.322} C_VEL
LIN {X 0,Y 233.021,Z 410.429,A -85,B 0,C 180,E1 -22719.375,E2 -22719.375} C_VEL
LIN {X 0,Y 227.984,Z 429.491,A -85,B 0,C 180,E1 -22718.764,E2 -22718.764} C_VEL
LIN {X 0,Y 227.133,Z 435.351,A -85,B 0,C 180,E1 -22718.788,E2 -22718.788} C_VEL
LIN {X 0,Y 224.074,Z 474.721,A -85,B 0,C 180,E1 -22719.875,E2 -22719.875} C_VEL
LIN {X 0,Y 221.746,Z 490.423,A -85,B 0,C 180,E1 -22720.567,E2 -22720.567} C_VEL
LIN {X 0,Y 218.704,Z 504.906,A -85,B 0,C 180,E1 -22721.485,E2 -22721.485} C_VEL
LIN {X 0,Y 214.978,Z 518.643,A -85,B 0,C 180,E1 -22722.646,E2 -22722.646} C_VEL
LIN {X 0,Y 210.624,Z 532.109,A -85,B 0,C 180,E1 -22724.161,E2 -22724.161} C_VEL
LIN {X 0,Y 205.677,Z 545.298,A -85,B 0,C 180,E1 -22726.077,E2 -22726.077} C_VEL
LIN {X 0,Y 200.025,Z 558.261,A -85,B 0,C 180,E1 -22728.458,E2 -22728.458} C_VEL
LIN {X 0,Y 194.972,Z 568.69,A -85,B 0,C 180,E1 -22730.891,E2 -22730.891} C_VEL
LIN {X 0,Y 189.866,Z 578.378,A -85,B 0,C 180,E1 -22733.684,E2 -22733.684} C_VEL
LIN {X 0,Y 184.689,Z 587.952,A -85,B 0,C 180,E1 -22737.185,E2 -22737.185} C_VEL
LIN {X 0,Y 180.234,Z 595.863,A -85,B 0,C 180,E1 -22740.83,E2 -22740.83} C_VEL
LIN {X 0,Y 175.942,Z 603.294,A -85,B 0,C 180,E1 -22745.203,E2 -22745.203} C_VEL
LIN {X 0,Y 172.672,Z 609.342,A -85,B 0,C 180,E1 -22749.895,E2 -22749.895} C_VEL
LIN {X 0,Y 171.024,Z 612.73,A -85,B 0,C 180,E1 -22753.284,E2 -22753.284} C_VEL
LIN {X 0,Y 169.507,Z 616.298,A -85,B 0,C 180,E1 -22758.037,E2 -22758.037} C_VEL
LIN {X 0,Y 168.927,Z 618.659,A -85,B 0,C 180,E1 -22762.831,E2 -22762.831} C_VEL
LIN {X 0,Y 168.928,Z 619.737,A -85,B 0,C 180,E1 -22766.841,E2 -22766.841} C_VEL
LIN {X 0,Y 169.089,Z 620.015,A -85,B 0,C 180,E1 -22770.001,E2 -22770.001} C_VEL
LIN {X 0,Y 168.929,Z 619.385,A -85,B 0,C 180,E1 -22774.774,E2 -22774.774} C_VEL
LIN {X 0,Y 169.126,Z 617.587,A -85,B 0,C 180,E1 -22779.569,E2 -22779.569} C_VEL
LIN {X 0,Y 170.098,Z 614.611,A -85,B 0,C 180,E1 -22784.355,E2 -22784.355} C_VEL
LIN {X 0,Y 172.12,Z 610.397,A -85,B 0,C 180,E1 -22789.067,E2 -22789.067} C_VEL
LIN {X 0,Y 175.014,Z 604.829,A -85,B 0,C 180,E1 -22793.678,E2 -22793.678} C_VEL
LIN {X 0,Y 178.982,Z 597.765,A -85,B 0,C 180,E1 -22798.113,E2 -22798.113} C_VEL
LIN {X 0,Y 183.334,Z 590.227,A -85,B 0,C 180,E1 -22801.811,E2 -22801.811} C_VEL
LIN {X 0,Y 188.332,Z 581.145,A -85,B 0,C 180,E1 -22805.34,E2 -22805.34} C_VEL
LIN {X 0,Y 194.068,Z 570.242,A -85,B 0,C 180,E1 -22808.661,E2 -22808.661} C_VEL
LIN {X 0,Y 199.523,Z 559.028,A -85,B 0,C 180,E1 -22811.336,E2 -22811.336} C_VEL
LIN {X 0,Y 205.064,Z 546.528,A -85,B 0,C 180,E1 -22813.673,E2 -22813.673} C_VEL
LIN {X 0,Y 210.098,Z 533.24,A -85,B 0,C 180,E1 -22815.646,E2 -22815.646} C_VEL
LIN {X 0,Y 214.391,Z 519.97,A -85,B 0,C 180,E1 -22817.181,E2 -22817.181} C_VEL
LIN {X 0,Y 218.09,Z 506.586,A -85,B 0,C 180,E1 -22818.352,E2 -22818.352} C_VEL
LIN {X 0,Y 221.326,Z 491.934,A -85,B 0,C 180,E1 -22819.301,E2 -22819.301} C_VEL
LIN {X 0,Y 223.595,Z 477.01,A -85,B 0,C 180,E1 -22820.007,E2 -22820.007} C_VEL
LIN {X 0,Y 225.401,Z 457.166,A -85,B 0,C 180,E1 -22820.588,E2 -22820.588} C_VEL
LIN {X 0,Y 229.509,Z 398.619,A -85,B 0,C 180,E1 -22822.189,E2 -22822.189} C_VEL
LIN {X 0,Y 224.513,Z 386.277,A -85,B 0,C 180,E1 -22824.502,E2 -22824.502} C_VEL
LIN {X 0,Y 219.125,Z 374.779,A -85,B 0,C 180,E1 -22827.175,E2 -22827.175} C_VEL
LIN {X 0,Y 213.961,Z 364.74,A -85,B 0,C 180,E1 -22830.007,E2 -22830.007} C_VEL
LIN {X 0,Y 209.775,Z 357.442,A -85,B 0,C 180,E1 -22832.548,E2 -22832.548} C_VEL
LIN {X 0,Y 207.873,Z 354.342,A -85,B 0,C 180,E1 -22833.796,E2 -22833.796} C_VEL
LIN {X 0,Y 204.833,Z 350.097,A -85,B 0,C 180,E1 -22835.908,E2 -22835.908} C_VEL
LIN {X 0,Y 201.631,Z 345.805,A -85,B 0,C 180,E1 -22838.398,E2 -22838.398} C_VEL
LIN {X 0,Y 198.786,Z 342.273,A -85,B 0,C 180,E1 -22840.912,E2 -22840.912} C_VEL
LIN {X 0,Y 197.815,Z 340.844,A -85,B 0,C 180,E1 -22841.888,E2 -22841.888} C_VEL
LIN {X 0,Y 195.306,Z 338.13,A -85,B 0,C 180,E1 -22844.605,E2 -22844.605} C_VEL
LIN {X 0,Y 194.017,Z 335.726,A -85,B 0,C 180,E1 -22846.382,E2 -22846.382} C_VEL
LIN {X 0,Y 191.518,Z 333.738,A -85,B 0,C 180,E1 -22850.229,E2 -22850.229} C_VEL
LIN {X 0,Y 190.019,Z 330.414,A -85,B 0,C 180,E1 -22854.296,E2 -22854.296} C_VEL
LIN {X 0,Y 189.622,Z 330.035,A -85,B 0,C 180,E1 -22855.749,E2 -22855.749} C_VEL
LIN {X 0,Y 189.152,Z 329.81,A -85,B 0,C 180,E1 -22862.13,E2 -22862.13} C_VEL
LIN {X 0,Y 190.02,Z 330.275,A -85,B 0,C 180,E1 -22866.237,E2 -22866.237} C_VEL
LIN {X 0,Y 191.111,Z 333.234,A -85,B 0,C 180,E1 -22869.526,E2 -22869.526} C_VEL
LIN {X 0,Y 193.208,Z 335.391,A -85,B 0,C 180,E1 -22873.141,E2 -22873.141} C_VEL
LIN {X 0,Y 194.159,Z 336.01,A -85,B 0,C 180,E1 -22874.41,E2 -22874.41} C_VEL
LIN {X 0,Y 196.188,Z 339.451,A -85,B 0,C 180,E1 -22877.034,E2 -22877.034} C_VEL
LIN {X 0,Y 198.392,Z 341.53,A -85,B 0,C 180,E1 -22879.263,E2 -22879.263} C_VEL
LIN {X 0,Y 200.851,Z 345.119,A -85,B 0,C 180,E1 -22881.556,E2 -22881.556} C_VEL
LIN {X 0,Y 202.318,Z 346.769,A -85,B 0,C 180,E1 -22882.75,E2 -22882.75} C_VEL
LIN {X 0,Y 205.839,Z 351.524,A -85,B 0,C 180,E1 -22885.399,E2 -22885.399} C_VEL
LIN {X 0,Y 209.38,Z 356.49,A -85,B 0,C 180,E1 -22887.757,E2 -22887.757} C_VEL
LIN {X 0,Y 214.154,Z 363.419,A -85,B 0,C 180,E1 -22890.576,E2 -22890.576} C_VEL
LIN {X 0,Y 220.583,Z 373.739,A -85,B 0,C 180,E1 -22893.922,E2 -22893.922} C_VEL
LIN {X 0,Y 227.115,Z 385.456,A -85,B 0,C 180,E1 -22896.937,E2 -22896.937} C_VEL
LIN {X 0,Y 229.978,Z 391.094,A -85,B 0,C 180,E1 -22898.168,E2 -22898.168} C_VEL
LIN {X 0,Y 224.834,Z 461.985,A -85,B 0,C 180,E1 -22900.119,E2 -22900.119} C_VEL
LIN {X 0,Y 222.734,Z 477.331,A -85,B 0,C 180,E1 -22900.773,E2 -22900.773} C_VEL
LIN {X 0,Y 219.802,Z 492.902,A -85,B 0,C 180,E1 -22901.805,E2 -22901.805} C_VEL
LIN {X 0,Y 216.296,Z 506.936,A -85,B 0,C 180,E1 -22903.063,E2 -22903.063} C_VEL
LIN {X 0,Y 212.348,Z 520.216,A -85,B 0,C 180,E1 -22904.635,E2 -22904.635} C_VEL
LIN {X 0,Y 207.299,Z 533.953,A -85,B 0,C 180,E1 -22906.642,E2 -22906.642} C_VEL
LIN {X 0,Y 202.064,Z 546.341,A -85,B 0,C 180,E1 -22908.966,E2 -22908.966} C_VEL
LIN {X 0,Y 197.08,Z 556.713,A -85,B 0,C 180,E1 -22911.385,E2 -22911.385} C_VEL
LIN {X 0,Y 192.322,Z 566.318,A -85,B 0,C 180,E1 -22914.218,E2 -22914.218} C_VEL
LIN {X 0,Y 187.71,Z 574.522,A -85,B 0,C 180,E1 -22917.118,E2 -22917.118} C_VEL
LIN {X 0,Y 183.038,Z 582.577,A -85,B 0,C 180,E1 -22920.687,E2 -22920.687} C_VEL
LIN {X 0,Y 178.135,Z 590.682,A -85,B 0,C 180,E1 -22925.371,E2 -22925.371} C_VEL
LIN {X 0,Y 174.569,Z 596.666,A -85,B 0,C 180,E1 -22929.988,E2 -22929.988} C_VEL
LIN {X 0,Y 172.532,Z 600.088,A -85,B 0,C 180,E1 -22933.431,E2 -22933.431} C_VEL
LIN {X 0,Y 170.624,Z 603.545,A -85,B 0,C 180,E1 -22938.114,E2 -22938.114} C_VEL
LIN {X 0,Y 169.582,Z 605.821,A -85,B 0,C 180,E1 -22942.857,E2 -22942.857} C_VEL
LIN {X 0,Y 169.17,Z 606.976,A -85,B 0,C 180,E1 -22947.618,E2 -22947.618} C_VEL
LIN {X 0,Y 169.169,Z 606.987,A -85,B 0,C 180,E1 -22952.38,E2 -22952.38} C_VEL
LIN {X 0,Y 169.581,Z 605.879,A -85,B 0,C 180,E1 -22957.141,E2 -22957.141} C_VEL
LIN {X 0,Y 170.617,Z 603.648,A -85,B 0,C 180,E1 -22961.884,E2 -22961.884} C_VEL
LIN {X 0,Y 172.457,Z 600.233,A -85,B 0,C 180,E1 -22966.574,E2 -22966.574} C_VEL
LIN {X 0,Y 175.3,Z 595.544,A -85,B 0,C 180,E1 -22971.149,E2 -22971.149} C_VEL
LIN {X 0,Y 178.927,Z 589.467,A -85,B 0,C 180,E1 -22975.598,E2 -22975.598} C_VEL
LIN {X 0,Y 183.573,Z 581.8,A -85,B 0,C 180,E1 -22979.847,E2 -22979.847} C_VEL
LIN {X 0,Y 188.319,Z 573.621,A -85,B 0,C 180,E1 -22983.398,E2 -22983.398} C_VEL
LIN {X 0,Y 193.258,Z 564.652,A -85,B 0,C 180,E1 -22986.482,E2 -22986.482} C_VEL
LIN {X 0,Y 197.852,Z 555.416,A -85,B 0,C 180,E1 -22989.086,E2 -22989.086} C_VEL
LIN {X 0,Y 203.38,Z 543.71,A -85,B 0,C 180,E1 -22991.697,E2 -22991.697} C_VEL
LIN {X 0,Y 208.175,Z 532.054,A -85,B 0,C 180,E1 -22993.794,E2 -22993.794} C_VEL
LIN {X 0,Y 212.674,Z 519.48,A -85,B 0,C 180,E1 -22995.611,E2 -22995.611} C_VEL
LIN {X 0,Y 216.85,Z 505.394,A -85,B 0,C 180,E1 -22997.223,E2 -22997.223} C_VEL
LIN {X 0,Y 220.222,Z 491.667,A -85,B 0,C 180,E1 -22998.413,E2 -22998.413} C_VEL
LIN {X 0,Y 222.951,Z 477.421,A -85,B 0,C 180,E1 -22999.329,E2 -22999.329} C_VEL
LIN {X 0,Y 224.929,Z 462.243,A -85,B 0,C 180,E1 -23000.016,E2 -23000.016} C_VEL
LIN {X 0,Y 230.162,Z 391.163,A -85,B 0,C 180,E1 -23001.952,E2 -23001.952} C_VEL
LIN {X 0,Y 223.707,Z 379.026,A -85,B 0,C 180,E1 -23004.798,E2 -23004.798} C_VEL
LIN {X 0,Y 217.723,Z 368.979,A -85,B 0,C 180,E1 -23007.726,E2 -23007.726} C_VEL
LIN {X 0,Y 212.427,Z 360.777,A -85,B 0,C 180,E1 -23010.641,E2 -23010.641} C_VEL
LIN {X 0,Y 207.896,Z 354.328,A -85,B 0,C 180,E1 -23013.457,E2 -23013.457} C_VEL
LIN {X 0,Y 204.845,Z 350.156,A -85,B 0,C 180,E1 -23015.588,E2 -23015.588} C_VEL
LIN {X 0,Y 201.729,Z 345.925,A -85,B 0,C 180,E1 -23018.039,E2 -23018.039} C_VEL
LIN {X 0,Y 198.934,Z 342.494,A -85,B 0,C 180,E1 -23020.524,E2 -23020.524} C_VEL
LIN {X 0,Y 198.109,Z 341.06,A -85,B 0,C 180,E1 -23021.38,E2 -23021.38} C_VEL
LIN {X 0,Y 195.621,Z 338.664,A -85,B 0,C 180,E1 -23024.034,E2 -23024.034} C_VEL
LIN {X 0,Y 194.122,Z 335.814,A -85,B 0,C 180,E1 -23026.122,E2 -23026.122} C_VEL
LIN {X 0,Y 191.541,Z 333.798,A -85,B 0,C 180,E1 -23030.229,E2 -23030.229} C_VEL
LIN {X 0,Y 189.947,Z 330.111,A -85,B 0,C 180,E1 -23035.224,E2 -23035.224} C_VEL
LIN {X 0,Y 189.394,Z 329.79,A -85,B 0,C 180,E1 -23040,E2 -23040} C_VEL
LIN {X 0,Y 190.076,Z 330.396,A -85,B 0,C 180,E1 -23044.872,E2 -23044.872} C_VEL
LIN {X 0,Y 191.918,Z 334.225,A -85,B 0,C 180,E1 -23050.017,E2 -23050.017} C_VEL
LIN {X 0,Y 194.314,Z 336.116,A -85,B 0,C 180,E1 -23053.664,E2 -23053.664} C_VEL
LIN {X 0,Y 196.396,Z 339.525,A -85,B 0,C 180,E1 -23056.368,E2 -23056.368} C_VEL
LIN {X 0,Y 198.349,Z 341.357,A -85,B 0,C 180,E1 -23058.369,E2 -23058.369} C_VEL
LIN {X 0,Y 200.999,Z 345.151,A -85,B 0,C 180,E1 -23060.867,E2 -23060.867} C_VEL
LIN {X 0,Y 202.369,Z 346.653,A -85,B 0,C 180,E1 -23061.988,E2 -23061.988} C_VEL
LIN {X 0,Y 206.065,Z 351.767,A -85,B 0,C 180,E1 -23064.796,E2 -23064.796} C_VEL
LIN {X 0,Y 208.918,Z 355.788,A -85,B 0,C 180,E1 -23066.722,E2 -23066.722} C_VEL
LIN {X 0,Y 213.793,Z 364.229,A -85,B 0,C 180,E1 -23069.747,E2 -23069.747} C_VEL
LIN {X 0,Y 219.824,Z 375.983,A -85,B 0,C 180,E1 -23073.059,E2 -23073.059} C_VEL
LIN {X 0,Y 225.089,Z 387.435,A -85,B 0,C 180,E1 -23075.661,E2 -23075.661} C_VEL
LIN {X 0,Y 229.673,Z 398.769,A -85,B 0,C 180,E1 -23077.779,E2 -23077.779} C_VEL
LIN {X 0,Y 227.133,Z 435.351,A -85,B 0,C 180,E1 -23078.788,E2 -23078.788} C_VEL
LIN {X 0,Y 226.3,Z 441.199,A -85,B 0,C 180,E1 -23078.813,E2 -23078.813} C_VEL
LIN {X 0,Y 221.294,Z 460.233,A -85,B 0,C 180,E1 -23078.163,E2 -23078.163} C_VEL
LIN {X 0,Y 220.414,Z 466.076,A -85,B 0,C 180,E1 -23078.192,E2 -23078.192} C_VEL
LIN {X 0,Y 218.658,Z 481.457,A -85,B 0,C 180,E1 -23078.72,E2 -23078.72} C_VEL
LIN {X 0,Y 215.891,Z 496.94,A -85,B 0,C 180,E1 -23079.548,E2 -23079.548} C_VEL
LIN {X 0,Y 212.305,Z 511.406,A -85,B 0,C 180,E1 -23080.598,E2 -23080.598} C_VEL
LIN {X 0,Y 207.949,Z 525.477,A -85,B 0,C 180,E1 -23081.968,E2 -23081.968} C_VEL
LIN {X 0,Y 202.83,Z 539.524,A -85,B 0,C 180,E1 -23083.795,E2 -23083.795} C_VEL
LIN {X 0,Y 197.291,Z 552.623,A -85,B 0,C 180,E1 -23086.003,E2 -23086.003} C_VEL
LIN {X 0,Y 191.306,Z 564.833,A -85,B 0,C 180,E1 -23088.605,E2 -23088.605} C_VEL
LIN {X 0,Y 185.869,Z 575.097,A -85,B 0,C 180,E1 -23091.4,E2 -23091.4} C_VEL
LIN {X 0,Y 179.973,Z 585.5,A -85,B 0,C 180,E1 -23095.023,E2 -23095.023} C_VEL
LIN {X 0,Y 174.662,Z 594.573,A -85,B 0,C 180,E1 -23099.135,E2 -23099.135} C_VEL
LIN {X 0,Y 170.467,Z 601.339,A -85,B 0,C 180,E1 -23103.032,E2 -23103.032} C_VEL
LIN {X 0,Y 166.763,Z 607.6,A -85,B 0,C 180,E1 -23107.711,E2 -23107.711} C_VEL
LIN {X 0,Y 164.143,Z 612.457,A -85,B 0,C 180,E1 -23112.561,E2 -23112.561} C_VEL
LIN {X 0,Y 162.506,Z 616.026,A -85,B 0,C 180,E1 -23117.513,E2 -23117.513} C_VEL
LIN {X 0,Y 161.865,Z 618.388,A -85,B 0,C 180,E1 -23122.517,E2 -23122.517} C_VEL
LIN {X 0,Y 161.864,Z 619.584,A -85,B 0,C 180,E1 -23127.513,E2 -23127.513} C_VEL
LIN {X 0,Y 161.995,Z 619.745,A -85,B 0,C 180,E1 -23130.001,E2 -23130.001} C_VEL
LIN {X 0,Y 161.839,Z 619.114,A -85,B 0,C 180,E1 -23134.984,E2 -23134.984} C_VEL
LIN {X 0,Y 162.085,Z 617.315,A -85,B 0,C 180,E1 -23139.989,E2 -23139.989} C_VEL
LIN {X 0,Y 163.172,Z 614.338,A -85,B 0,C 180,E1 -23144.978,E2 -23144.978} C_VEL
LIN {X 0,Y 165.341,Z 610.123,A -85,B 0,C 180,E1 -23149.881,E2 -23149.881} C_VEL
LIN {X 0,Y 168.459,Z 604.554,A -85,B 0,C 180,E1 -23154.659,E2 -23154.659} C_VEL
LIN {X 0,Y 172.686,Z 597.49,A -85,B 0,C 180,E1 -23159.235,E2 -23159.235} C_VEL
LIN {X 0,Y 177.277,Z 589.951,A -85,B 0,C 180,E1 -23163.033,E2 -23163.033} C_VEL
LIN {X 0,Y 182.521,Z 580.87,A -85,B 0,C 180,E1 -23166.645,E2 -23166.645} C_VEL
LIN {X 0,Y 188.53,Z 569.967,A -85,B 0,C 180,E1 -23170.021,E2 -23170.021} C_VEL
LIN {X 0,Y 194.23,Z 558.754,A -85,B 0,C 180,E1 -23172.724,E2 -23172.724} C_VEL
LIN {X 0,Y 199.777,Z 546.661,A -85,B 0,C 180,E1 -23175.015,E2 -23175.015} C_VEL
LIN {X 0,Y 204.632,Z 534.396,A -85,B 0,C 180,E1 -23176.873,E2 -23176.873} C_VEL
LIN {X 0,Y 209.067,Z 521.466,A -85,B 0,C 180,E1 -23178.415,E2 -23178.415} C_VEL
LIN {X 0,Y 213.134,Z 507.438,A -85,B 0,C 180,E1 -23179.69,E2 -23179.69} C_VEL
LIN {X 0,Y 216.602,Z 492.417,A -85,B 0,C 180,E1 -23180.684,E2 -23180.684} C_VEL
LIN {X 0,Y 219.014,Z 477.406,A -85,B 0,C 180,E1 -23181.403,E2 -23181.403} C_VEL
LIN {X 0,Y 220.922,Z 457.399,A -85,B 0,C 180,E1 -23181.996,E2 -23181.996} C_VEL
LIN {X 0,Y 224.996,Z 401.182,A -85,B 0,C 180,E1 -23183.545,E2 -23183.545} C_VEL
LIN {X 0,Y 220.635,Z 390.222,A -85,B 0,C 180,E1 -23185.701,E2 -23185.701} C_VEL
LIN {X 0,Y 215.526,Z 378.928,A -85,B 0,C 180,E1 -23188.414,E2 -23188.414} C_VEL
LIN {X 0,Y 210.563,Z 369.107,A -85,B 0,C 180,E1 -23191.328,E2 -23191.328} C_VEL
LIN {X 0,Y 205.992,Z 360.883,A -85,B 0,C 180,E1 -23194.35,E2 -23194.35} C_VEL
LIN {X 0,Y 202.468,Z 356.009,A -85,B 0,C 180,E1 -23196.906,E2 -23196.906} C_VEL
LIN {X 0,Y 199.765,Z 352.249,A -85,B 0,C 180,E1 -23199.133,E2 -23199.133} C_VEL
LIN {X 0,Y 196.831,Z 348.239,A -85,B 0,C 180,E1 -23201.912,E2 -23201.912} C_VEL
LIN {X 0,Y 193.549,Z 344.186,A -85,B 0,C 180,E1 -23205.678,E2 -23205.678} C_VEL
LIN {X 0,Y 192.775,Z 342.639,A -85,B 0,C 180,E1 -23206.829,E2 -23206.829} C_VEL
LIN {X 0,Y 190.391,Z 340.569,A -85,B 0,C 180,E1 -23210.706,E2 -23210.706} C_VEL
LIN {X 0,Y 188.901,Z 337.131,A -85,B 0,C 180,E1 -23215.198,E2 -23215.198} C_VEL
LIN {X 0,Y 188.206,Z 336.743,A -85,B 0,C 180,E1 -23220,E2 -23220} C_VEL
LIN {X 0,Y 189.06,Z 337.407,A -85,B 0,C 180,E1 -23226.001,E2 -23226.001} C_VEL
LIN {X 0,Y 190.453,Z 340.764,A -85,B 0,C 180,E1 -23230.028,E2 -23230.028} C_VEL
LIN {X 0,Y 192.912,Z 342.942,A -85,B 0,C 180,E1 -23233.967,E2 -23233.967} C_VEL
LIN {X 0,Y 194.902,Z 346.311,A -85,B 0,C 180,E1 -23236.632,E2 -23236.632} C_VEL
LIN {X 0,Y 196.836,Z 348.24,A -85,B 0,C 180,E1 -23238.673,E2 -23238.673} C_VEL
LIN {X 0,Y 199.437,Z 351.955,A -85,B 0,C 180,E1 -23241.174,E2 -23241.174} C_VEL
LIN {X 0,Y 200.457,Z 353.162,A -85,B 0,C 180,E1 -23242.04,E2 -23242.04} C_VEL
LIN {X 0,Y 203.983,Z 358.13,A -85,B 0,C 180,E1 -23244.817,E2 -23244.817} C_VEL
LIN {X 0,Y 207.194,Z 362.768,A -85,B 0,C 180,E1 -23247.048,E2 -23247.048} C_VEL
LIN {X 0,Y 211.75,Z 369.553,A -85,B 0,C 180,E1 -23249.858,E2 -23249.858} C_VEL
LIN {X 0,Y 217.692,Z 379.457,A -85,B 0,C 180,E1 -23253.103,E2 -23253.103} C_VEL
LIN {X 0,Y 223.614,Z 390.352,A -85,B 0,C 180,E1 -23255.979,E2 -23255.979} C_VEL
LIN {X 0,Y 225.465,Z 394.059,A -85,B 0,C 180,E1 -23256.823,E2 -23256.823} C_VEL
LIN {X 0,Y 220.356,Z 462.115,A -85,B 0,C 180,E1 -23258.707,E2 -23258.707} C_VEL
LIN {X 0,Y 218.308,Z 476.809,A -85,B 0,C 180,E1 -23259.328,E2 -23259.328} C_VEL
LIN {X 0,Y 215.407,Z 491.894,A -85,B 0,C 180,E1 -23260.3,E2 -23260.3} C_VEL
LIN {X 0,Y 211.664,Z 506.698,A -85,B 0,C 180,E1 -23261.611,E2 -23261.611} C_VEL
LIN {X 0,Y 207.431,Z 520.491,A -85,B 0,C 180,E1 -23263.242,E2 -23263.242} C_VEL
LIN {X 0,Y 202.203,Z 534.227,A -85,B 0,C 180,E1 -23265.263,E2 -23265.263} C_VEL
LIN {X 0,Y 196.768,Z 546.615,A -85,B 0,C 180,E1 -23267.609,E2 -23267.609} C_VEL
LIN {X 0,Y 191.57,Z 556.987,A -85,B 0,C 180,E1 -23270.057,E2 -23270.057} C_VEL
LIN {X 0,Y 186.579,Z 566.592,A -85,B 0,C 180,E1 -23272.936,E2 -23272.936} C_VEL
LIN {X 0,Y 181.767,Z 574.796,A -85,B 0,C 180,E1 -23275.898,E2 -23275.898} C_VEL
LIN {X 0,Y 176.87,Z 582.85,A -85,B 0,C 180,E1 -23279.559,E2 -23279.559} C_VEL
LIN {X 0,Y 172.031,Z 590.418,A -85,B 0,C 180,E1 -23283.997,E2 -23283.997} C_VEL
LIN {X 0,Y 167.901,Z 596.938,A -85,B 0,C 180,E1 -23289.157,E2 -23289.157} C_VEL
LIN {X 0,Y 165.694,Z 600.362,A -85,B 0,C 180,E1 -23292.727,E2 -23292.727} C_VEL
LIN {X 0,Y 163.672,Z 603.817,A -85,B 0,C 180,E1 -23297.601,E2 -23297.601} C_VEL
LIN {X 0,Y 162.541,Z 606.092,A -85,B 0,C 180,E1 -23302.546,E2 -23302.546} C_VEL
LIN {X 0,Y 162.085,Z 607.246,A -85,B 0,C 180,E1 -23307.514,E2 -23307.514} C_VEL
LIN {X 0,Y 162.085,Z 607.257,A -85,B 0,C 180,E1 -23312.484,E2 -23312.484} C_VEL
LIN {X 0,Y 162.54,Z 606.149,A -85,B 0,C 180,E1 -23317.452,E2 -23317.452} C_VEL
LIN {X 0,Y 163.664,Z 603.918,A -85,B 0,C 180,E1 -23322.397,E2 -23322.397} C_VEL
LIN {X 0,Y 165.623,Z 600.504,A -85,B 0,C 180,E1 -23327.279,E2 -23327.279} C_VEL
LIN {X 0,Y 168.673,Z 595.815,A -85,B 0,C 180,E1 -23332.023,E2 -23332.023} C_VEL
LIN {X 0,Y 172.527,Z 589.737,A -85,B 0,C 180,E1 -23336.62,E2 -23336.62} C_VEL
LIN {X 0,Y 177.426,Z 582.07,A -85,B 0,C 180,E1 -23340.992,E2 -23340.992} C_VEL
LIN {X 0,Y 182.414,Z 573.891,A -85,B 0,C 180,E1 -23344.629,E2 -23344.629} C_VEL
LIN {X 0,Y 187.332,Z 565.361,A -85,B 0,C 180,E1 -23347.632,E2 -23347.632} C_VEL
LIN {X 0,Y 192.371,Z 555.684,A -85,B 0,C 180,E1 -23350.425,E2 -23350.425} C_VEL
LIN {X 0,Y 198.127,Z 543.977,A -85,B 0,C 180,E1 -23353.065,E2 -23353.065} C_VEL
LIN {X 0,Y 203.116,Z 532.32,A -85,B 0,C 180,E1 -23355.178,E2 -23355.178} C_VEL
LIN {X 0,Y 207.774,Z 519.745,A -85,B 0,C 180,E1 -23357.009,E2 -23357.009} C_VEL
LIN {X 0,Y 211.663,Z 507.205,A -85,B 0,C 180,E1 -23358.483,E2 -23358.483} C_VEL
LIN {X 0,Y 215.298,Z 493.215,A -85,B 0,C 180,E1 -23359.731,E2 -23359.731} C_VEL
LIN {X 0,Y 218.263,Z 478.565,A -85,B 0,C 180,E1 -23360.689,E2 -23360.689} C_VEL
LIN {X 0,Y 220.332,Z 463.548,A -85,B 0,C 180,E1 -23361.387,E2 -23361.387} C_VEL
LIN {X 0,Y 223.906,Z 417.534,A -85,B 0,C 180,E1 -23362.67,E2 -23362.67} C_VEL
LIN {X 0,Y 225.633,Z 394.174,A -85,B 0,C 180,E1 -23363.302,E2 -23363.302} C_VEL
LIN {X 0,Y 220.016,Z 383.416,A -85,B 0,C 180,E1 -23365.945,E2 -23365.945} C_VEL
LIN {X 0,Y 214.615,Z 374.176,A -85,B 0,C 180,E1 -23368.746,E2 -23368.746} C_VEL
LIN {X 0,Y 209.967,Z 366.741,A -85,B 0,C 180,E1 -23371.446,E2 -23371.446} C_VEL
LIN {X 0,Y 205.614,Z 360.39,A -85,B 0,C 180,E1 -23374.288,E2 -23374.288} C_VEL
LIN {X 0,Y 203.007,Z 356.661,A -85,B 0,C 180,E1 -23376.201,E2 -23376.201} C_VEL
LIN {X 0,Y 199.862,Z 352.356,A -85,B 0,C 180,E1 -23378.782,E2 -23378.782} C_VEL
LIN {X 0,Y 197.146,Z 348.738,A -85,B 0,C 180,E1 -23381.354,E2 -23381.354} C_VEL
LIN {X 0,Y 196.391,Z 347.646,A -85,B 0,C 180,E1 -23382.156,E2 -23382.156} C_VEL
LIN {X 0,Y 193.976,Z 344.921,A -85,B 0,C 180,E1 -23384.949,E2 -23384.949} C_VEL
LIN {X 0,Y 192.701,Z 342.644,A -85,B 0,C 180,E1 -23386.824,E2 -23386.824} C_VEL
LIN {X 0,Y 190.267,Z 340.348,A -85,B 0,C 180,E1 -23391.091,E2 -23391.091} C_VEL
LIN {X 0,Y 189.065,Z 337.155,A -85,B 0,C 180,E1 -23395.28,E2 -23395.28} C_VEL
LIN {X 0,Y 188.529,Z 336.838,A -85,B 0,C 180,E1 -23400,E2 -23400} C_VEL
LIN {X 0,Y 189.117,Z 337.383,A -85,B 0,C 180,E1 -23404.529,E2 -23404.529} C_VEL
LIN {X 0,Y 190.866,Z 341.168,A -85,B 0,C 180,E1 -23409.704,E2 -23409.704} C_VEL
LIN {X 0,Y 193.028,Z 342.976,A -85,B 0,C 180,E1 -23413.153,E2 -23413.153} C_VEL
LIN {X 0,Y 195.312,Z 346.598,A -85,B 0,C 180,E1 -23416.193,E2 -23416.193} C_VEL
LIN {X 0,Y 196.849,Z 348.125,A -85,B 0,C 180,E1 -23417.823,E2 -23417.823} C_VEL
LIN {X 0,Y 199.614,Z 352.009,A -85,B 0,C 180,E1 -23420.505,E2 -23420.505} C_VEL
LIN {X 0,Y 200.768,Z 353.475,A -85,B 0,C 180,E1 -23421.497,E2 -23421.497} C_VEL
LIN {X 0,Y 204.031,Z 358.065,A -85,B 0,C 180,E1 -23424.077,E2 -23424.077} C_VEL
LIN {X 0,Y 206.769,Z 362.139,A -85,B 0,C 180,E1 -23426.02,E2 -23426.02} C_VEL
LIN {X 0,Y 211.121,Z 369.969,A -85,B 0,C 180,E1 -23428.861,E2 -23428.861} C_VEL
LIN {X 0,Y 216.731,Z 381.285,A -85,B 0,C 180,E1 -23432.116,E2 -23432.116} C_VEL
LIN {X 0,Y 221.816,Z 392.745,A -85,B 0,C 180,E1 -23434.772,E2 -23434.772} C_VEL
LIN {X 0,Y 225.209,Z 401.407,A -85,B 0,C 180,E1 -23436.441,E2 -23436.441} C_VEL
LIN {X 0,Y 220.414,Z 466.076,A -85,B 0,C 180,E1 -23438.192,E2 -23438.192} C_VEL
LIN {X 0,Y 219.472,Z 471.896,A -85,B 0,C 180,E1 -23438.232,E2 -23438.232} C_VEL
LIN {X 0,Y 216.532,Z 481.312,A -85,B 0,C 180,E1 -23438.011,E2 -23438.011} C_VEL
LIN {X 0,Y 213.157,Z 490.621,A -85,B 0,C 180,E1 -23437.867,E2 -23437.867} C_VEL
LIN {X 0,Y 211.532,Z 496.275,A -85,B 0,C 180,E1 -23438.041,E2 -23438.041} C_VEL
LIN {X 0,Y 207.754,Z 511.142,A -85,B 0,C 180,E1 -23439.111,E2 -23439.111} C_VEL
LIN {X 0,Y 203.256,Z 525.211,A -85,B 0,C 180,E1 -23440.476,E2 -23440.476} C_VEL
LIN {X 0,Y 198.209,Z 538.61,A -85,B 0,C 180,E1 -23442.206,E2 -23442.206} C_VEL
LIN {X 0,Y 192.743,Z 551.216,A -85,B 0,C 180,E1 -23444.31,E2 -23444.31} C_VEL
LIN {X 0,Y 187.006,Z 562.658,A -85,B 0,C 180,E1 -23446.697,E2 -23446.697} C_VEL
LIN {X 0,Y 181.251,Z 573.191,A -85,B 0,C 180,E1 -23449.499,E2 -23449.499} C_VEL
LIN {X 0,Y 175.985,Z 582.137,A -85,B 0,C 180,E1 -23452.483,E2 -23452.483} C_VEL
LIN {X 0,Y 170.569,Z 590.958,A -85,B 0,C 180,E1 -23456.205,E2 -23456.205} C_VEL
LIN {X 0,Y 166.511,Z 597.355,A -85,B 0,C 180,E1 -23459.571,E2 -23459.571} C_VEL
LIN {X 0,Y 161.976,Z 604.382,A -85,B 0,C 180,E1 -23464.286,E2 -23464.286} C_VEL
LIN {X 0,Y 158.605,Z 609.923,A -85,B 0,C 180,E1 -23469.239,E2 -23469.239} C_VEL
LIN {X 0,Y 156.269,Z 614.123,A -85,B 0,C 180,E1 -23474.346,E2 -23474.346} C_VEL
LIN {X 0,Y 155.034,Z 617.082,A -85,B 0,C 180,E1 -23479.554,E2 -23479.554} C_VEL
LIN {X 0,Y 154.732,Z 618.859,A -85,B 0,C 180,E1 -23484.789,E2 -23484.789} C_VEL
LIN {X 0,Y 154.904,Z 619.474,A -85,B 0,C 180,E1 -23490.001,E2 -23490.001} C_VEL
LIN {X 0,Y 154.732,Z 618.842,A -85,B 0,C 180,E1 -23495.213,E2 -23495.213} C_VEL
LIN {X 0,Y 155.034,Z 617.042,A -85,B 0,C 180,E1 -23500.448,E2 -23500.448} C_VEL
LIN {X 0,Y 156.269,Z 614.064,A -85,B 0,C 180,E1 -23505.656,E2 -23505.656} C_VEL
LIN {X 0,Y 158.606,Z 609.848,A -85,B 0,C 180,E1 -23510.763,E2 -23510.763} C_VEL
LIN {X 0,Y 161.959,Z 604.279,A -85,B 0,C 180,E1 -23515.719,E2 -23515.719} C_VEL
LIN {X 0,Y 166.478,Z 597.216,A -85,B 0,C 180,E1 -23520.438,E2 -23520.438} C_VEL
LIN {X 0,Y 171.317,Z 589.677,A -85,B 0,C 180,E1 -23524.339,E2 -23524.339} C_VEL
LIN {X 0,Y 176.815,Z 580.594,A -85,B 0,C 180,E1 -23528.033,E2 -23528.033} C_VEL
LIN {X 0,Y 183.111,Z 569.692,A -85,B 0,C 180,E1 -23531.46,E2 -23531.46} C_VEL
LIN {X 0,Y 188.014,Z 560.439,A -85,B 0,C 180,E1 -23533.753,E2 -23533.753} C_VEL
LIN {X 0,Y 193.786,Z 548.552,A -85,B 0,C 180,E1 -23536.122,E2 -23536.122} C_VEL
LIN {X 0,Y 199.261,Z 535.552,A -85,B 0,C 180,E1 -23538.168,E2 -23538.168} C_VEL
LIN {X 0,Y 204.402,Z 521.188,A -85,B 0,C 180,E1 -23539.911,E2 -23539.911} C_VEL
LIN {X 0,Y 208.622,Z 507.162,A -85,B 0,C 180,E1 -23541.173,E2 -23541.173} C_VEL
LIN {X 0,Y 212.181,Z 492.137,A -85,B 0,C 180,E1 -23542.166,E2 -23542.166} C_VEL
LIN {X 0,Y 214.699,Z 476.802,A -85,B 0,C 180,E1 -23542.896,E2 -23542.896} C_VEL
LIN {X 0,Y 216.676,Z 456.288,A -85,B 0,C 180,E1 -23543.502,E2 -23543.502} C_VEL
LIN {X 0,Y 220.645,Z 403.826,A -85,B 0,C 180,E1 -23544.941,E2 -23544.941} C_VEL
LIN {X 0,Y 216.41,Z 392.987,A -85,B 0,C 180,E1 -23547.193,E2 -23547.193} C_VEL
LIN {X 0,Y 211.456,Z 381.919,A -85,B 0,C 180,E1 -23550.036,E2 -23550.036} C_VEL
LIN {X 0,Y 206.983,Z 372.983,A -85,B 0,C 180,E1 -23552.885,E2 -23552.885} C_VEL
LIN {X 0,Y 203.549,Z 366.73,A -85,B 0,C 180,E1 -23555.319,E2 -23555.319} C_VEL
LIN {X 0,Y 200.723,Z 362.592,A -85,B 0,C 180,E1 -23557.483,E2 -23557.483} C_VEL
LIN {X 0,Y 197.938,Z 358.654,A -85,B 0,C 180,E1 -23559.882,E2 -23559.882} C_VEL
LIN {X 0,Y 194.772,Z 354.212,A -85,B 0,C 180,E1 -23563.087,E2 -23563.087} C_VEL
LIN {X 0,Y 192.294,Z 351.06,A -85,B 0,C 180,E1 -23566.123,E2 -23566.123} C_VEL
LIN {X 0,Y 191.549,Z 349.525,A -85,B 0,C 180,E1 -23567.283,E2 -23567.283} C_VEL
LIN {X 0,Y 189.158,Z 347.251,A -85,B 0,C 180,E1 -23571.453,E2 -23571.453} C_VEL
LIN {X 0,Y 188.041,Z 344.164,A -85,B 0,C 180,E1 -23575.176,E2 -23575.176} C_VEL
LIN {X 0,Y 187.343,Z 343.772,A -85,B 0,C 180,E1 -23580,E2 -23580} C_VEL
LIN {X 0,Y 188.077,Z 344.418,A -85,B 0,C 180,E1 -23585.629,E2 -23585.629} C_VEL
LIN {X 0,Y 189.683,Z 348.067,A -85,B 0,C 180,E1 -23590.272,E2 -23590.272} C_VEL
LIN {X 0,Y 191.676,Z 349.874,A -85,B 0,C 180,E1 -23593.518,E2 -23593.518} C_VEL
LIN {X 0,Y 193.823,Z 353.386,A -85,B 0,C 180,E1 -23596.456,E2 -23596.456} C_VEL
LIN {X 0,Y 195.378,Z 355.07,A -85,B 0,C 180,E1 -23598.16,E2 -23598.16} C_VEL
LIN {X 0,Y 198.172,Z 358.924,A -85,B 0,C 180,E1 -23600.908,E2 -23600.908} C_VEL
LIN {X 0,Y 202.007,Z 364.49,A -85,B 0,C 180,E1 -23604.114,E2 -23604.114} C_VEL
LIN {X 0,Y 205.046,Z 368.999,A -85,B 0,C 180,E1 -23606.324,E2 -23606.324} C_VEL
LIN {X 0,Y 209.877,Z 376.561,A -85,B 0,C 180,E1 -23609.431,E2 -23609.431} C_VEL
LIN {X 0,Y 215.046,Z 385.539,A -85,B 0,C 180,E1 -23612.37,E2 -23612.37} C_VEL
LIN {X 0,Y 220.297,Z 395.467,A -85,B 0,C 180,E1 -23615.047,E2 -23615.047} C_VEL
LIN {X 0,Y 221.077,Z 397.099,A -85,B 0,C 180,E1 -23615.427,E2 -23615.427} C_VEL
LIN {X 0,Y 215.991,Z 462.427,A -85,B 0,C 180,E1 -23617.24,E2 -23617.24} C_VEL
LIN {X 0,Y 213.761,Z 477.894,A -85,B 0,C 180,E1 -23617.9,E2 -23617.9} C_VEL
LIN {X 0,Y 210.628,Z 493.458,A -85,B 0,C 180,E1 -23618.933,E2 -23618.933} C_VEL
LIN {X 0,Y 206.848,Z 507.612,A -85,B 0,C 180,E1 -23620.208,E2 -23620.208} C_VEL
LIN {X 0,Y 202.642,Z 520.766,A -85,B 0,C 180,E1 -23621.783,E2 -23621.783} C_VEL
LIN {X 0,Y 197.227,Z 534.501,A -85,B 0,C 180,E1 -23623.812,E2 -23623.812} C_VEL
LIN {X 0,Y 191.592,Z 546.888,A -85,B 0,C 180,E1 -23626.18,E2 -23626.18} C_VEL
LIN {X 0,Y 186.164,Z 557.262,A -85,B 0,C 180,E1 -23628.649,E2 -23628.649} C_VEL
LIN {X 0,Y 180.933,Z 566.867,A -85,B 0,C 180,E1 -23631.574,E2 -23631.574} C_VEL
LIN {X 0,Y 175.162,Z 576.287,A -85,B 0,C 180,E1 -23635.126,E2 -23635.126} C_VEL
LIN {X 0,Y 170.066,Z 584.121,A -85,B 0,C 180,E1 -23638.897,E2 -23638.897} C_VEL
LIN {X 0,Y 165.414,Z 591.02,A -85,B 0,C 180,E1 -23643.156,E2 -23643.156} C_VEL
LIN {X 0,Y 161.273,Z 597.21,A -85,B 0,C 180,E1 -23648.257,E2 -23648.257} C_VEL
LIN {X 0,Y 158.888,Z 600.635,A -85,B 0,C 180,E1 -23651.962,E2 -23651.962} C_VEL
LIN {X 0,Y 156.744,Z 604.088,A -85,B 0,C 180,E1 -23657.044,E2 -23657.044} C_VEL
LIN {X 0,Y 155.496,Z 606.363,A -85,B 0,C 180,E1 -23662.206,E2 -23662.206} C_VEL
LIN {X 0,Y 154.993,Z 607.516,A -85,B 0,C 180,E1 -23667.4,E2 -23667.4} C_VEL
LIN {X 0,Y 154.992,Z 607.528,A -85,B 0,C 180,E1 -23672.598,E2 -23672.598} C_VEL
LIN {X 0,Y 155.495,Z 606.419,A -85,B 0,C 180,E1 -23677.792,E2 -23677.792} C_VEL
LIN {X 0,Y 156.733,Z 604.188,A -85,B 0,C 180,E1 -23682.955,E2 -23682.955} C_VEL
LIN {X 0,Y 158.82,Z 600.775,A -85,B 0,C 180,E1 -23688.043,E2 -23688.043} C_VEL
LIN {X 0,Y 162.087,Z 596.085,A -85,B 0,C 180,E1 -23692.968,E2 -23692.968} C_VEL
LIN {X 0,Y 166.184,Z 590.007,A -85,B 0,C 180,E1 -23697.722,E2 -23697.722} C_VEL
LIN {X 0,Y 171.35,Z 582.34,A -85,B 0,C 180,E1 -23702.221,E2 -23702.221} C_VEL
LIN {X 0,Y 176.611,Z 574.159,A -85,B 0,C 180,E1 -23705.94,E2 -23705.94} C_VEL
LIN {X 0,Y 181.605,Z 565.86,A -85,B 0,C 180,E1 -23708.927,E2 -23708.927} C_VEL
LIN {X 0,Y 187.026,Z 555.952,A -85,B 0,C 180,E1 -23711.835,E2 -23711.835} C_VEL
LIN {X 0,Y 192.99,Z 544.245,A -85,B 0,C 180,E1 -23714.507,E2 -23714.507} C_VEL
LIN {X 0,Y 198.18,Z 532.586,A -85,B 0,C 180,E1 -23716.633,E2 -23716.633} C_VEL
LIN {X 0,Y 203.005,Z 520.01,A -85,B 0,C 180,E1 -23718.473,E2 -23718.473} C_VEL
LIN {X 0,Y 207.318,Z 506.525,A -85,B 0,C 180,E1 -23720.037,E2 -23720.037} C_VEL
LIN {X 0,Y 211.091,Z 492.189,A -85,B 0,C 180,E1 -23721.289,E2 -23721.289} C_VEL
LIN {X 0,Y 214.07,Z 477.309,A -85,B 0,C 180,E1 -23722.246,E2 -23722.246} C_VEL
LIN {X 0,Y 216.118,Z 462.613,A -85,B 0,C 180,E1 -23722.897,E2 -23722.897} C_VEL
LIN {X 0,Y 221.284,Z 397.223,A -85,B 0,C 180,E1 -23724.686,E2 -23724.686} C_VEL
LIN {X 0,Y 215.447,Z 386.041,A -85,B 0,C 180,E1 -23727.643,E2 -23727.643} C_VEL
LIN {X 0,Y 209.839,Z 376.426,A -85,B 0,C 180,E1 -23730.832,E2 -23730.832} C_VEL
LIN {X 0,Y 206.037,Z 370.382,A -85,B 0,C 180,E1 -23733.267,E2 -23733.267} C_VEL
LIN {X 0,Y 203.19,Z 366.175,A -85,B 0,C 180,E1 -23735.275,E2 -23735.275} C_VEL
LIN {X 0,Y 200.708,Z 362.562,A -85,B 0,C 180,E1 -23737.209,E2 -23737.209} C_VEL
LIN {X 0,Y 198.089,Z 358.821,A -85,B 0,C 180,E1 -23739.491,E2 -23739.491} C_VEL
LIN {X 0,Y 195.401,Z 354.981,A -85,B 0,C 180,E1 -23742.198,E2 -23742.198} C_VEL
LIN {X 0,Y 192.418,Z 351.22,A -85,B 0,C 180,E1 -23745.828,E2 -23745.828} C_VEL
LIN {X 0,Y 191.49,Z 349.539,A -85,B 0,C 180,E1 -23747.278,E2 -23747.278} C_VEL
LIN {X 0,Y 189.23,Z 347.249,A -85,B 0,C 180,E1 -23751.456,E2 -23751.456} C_VEL
LIN {X 0,Y 188.092,Z 344.188,A -85,B 0,C 180,E1 -23755.714,E2 -23755.714} C_VEL
LIN {X 0,Y 187.664,Z 343.882,A -85,B 0,C 180,E1 -23760,E2 -23760} C_VEL
LIN {X 0,Y 188.183,Z 344.425,A -85,B 0,C 180,E1 -23764.283,E2 -23764.283} C_VEL
LIN {X 0,Y 190.004,Z 348.296,A -85,B 0,C 180,E1 -23769.748,E2 -23769.748} C_VEL
LIN {X 0,Y 191.802,Z 349.869,A -85,B 0,C 180,E1 -23772.7,E2 -23772.7} C_VEL
LIN {X 0,Y 194.016,Z 353.424,A -85,B 0,C 180,E1 -23775.764,E2 -23775.764} C_VEL
LIN {X 0,Y 195.472,Z 355.051,A -85,B 0,C 180,E1 -23777.385,E2 -23777.385} C_VEL
LIN {X 0,Y 198.32,Z 358.964,A -85,B 0,C 180,E1 -23780.213,E2 -23780.213} C_VEL
LIN {X 0,Y 202.028,Z 364.379,A -85,B 0,C 180,E1 -23783.344,E2 -23783.344} C_VEL
LIN {X 0,Y 204.573,Z 368.334,A -85,B 0,C 180,E1 -23785.244,E2 -23785.244} C_VEL
LIN {X 0,Y 208.672,Z 376.042,A -85,B 0,C 180,E1 -23788.064,E2 -23788.064} C_VEL
LIN {X 0,Y 213.759,Z 386.713,A -85,B 0,C 180,E1 -23791.18,E2 -23791.18} C_VEL
LIN {X 0,Y 218.896,Z 398.803,A -85,B 0,C 180,E1 -23794.012,E2 -23794.012} C_VEL
LIN {X 0,Y 220.82,Z 403.89,A -85,B 0,C 180,E1 -23795.021,E2 -23795.021} C_VEL
LIN {X 0,Y 215.37,Z 473.362,A -85,B 0,C 180,E1 -23796.946,E2 -23796.946} C_VEL
LIN {X 0,Y 212.942,Z 489.138,A -85,B 0,C 180,E1 -23797.619,E2 -23797.619} C_VEL
LIN {X 0,Y 211.532,Z 496.275,A -85,B 0,C 180,E1 -23798.041,E2 -23798.041} C_VEL
LIN {X 0,Y 209.732,Z 501.872,A -85,B 0,C 180,E1 -23798.228,E2 -23798.228} C_VEL
LIN {X 0,Y 205.414,Z 510.823,A -85,B 0,C 180,E1 -23798.268,E2 -23798.268} C_VEL
LIN {X 0,Y 200.902,Z 519.681,A -85,B 0,C 180,E1 -23798.487,E2 -23798.487} C_VEL
LIN {X 0,Y 198.745,Z 524.871,A -85,B 0,C 180,E1 -23798.91,E2 -23798.91} C_VEL
LIN {X 0,Y 193.048,Z 539.381,A -85,B 0,C 180,E1 -23800.797,E2 -23800.797} C_VEL
LIN {X 0,Y 187.28,Z 552.085,A -85,B 0,C 180,E1 -23802.966,E2 -23802.966} C_VEL
LIN {X 0,Y 180.823,Z 564.293,A -85,B 0,C 180,E1 -23805.606,E2 -23805.606} C_VEL
LIN {X 0,Y 174.903,Z 574.556,A -85,B 0,C 180,E1 -23808.472,E2 -23808.472} C_VEL
LIN {X 0,Y 168.74,Z 584.431,A -85,B 0,C 180,E1 -23812.007,E2 -23812.007} C_VEL
LIN {X 0,Y 163.208,Z 592.944,A -85,B 0,C 180,E1 -23815.959,E2 -23815.959} C_VEL
LIN {X 0,Y 157.815,Z 600.795,A -85,B 0,C 180,E1 -23820.67,E2 -23820.67} C_VEL
LIN {X 0,Y 153.566,Z 607.055,A -85,B 0,C 180,E1 -23825.678,E2 -23825.678} C_VEL
LIN {X 0,Y 150.493,Z 611.911,A -85,B 0,C 180,E1 -23830.921,E2 -23830.921} C_VEL
LIN {X 0,Y 148.53,Z 615.48,A -85,B 0,C 180,E1 -23836.316,E2 -23836.316} C_VEL
LIN {X 0,Y 147.717,Z 617.844,A -85,B 0,C 180,E1 -23841.795,E2 -23841.795} C_VEL
LIN {X 0,Y 147.675,Z 619.043,A -85,B 0,C 180,E1 -23847.274,E2 -23847.274} C_VEL
LIN {X 0,Y 147.804,Z 619.204,A -85,B 0,C 180,E1 -23850.001,E2 -23850.001} C_VEL
LIN {X 0,Y 147.635,Z 618.57,A -85,B 0,C 180,E1 -23855.465,E2 -23855.465} C_VEL
LIN {X 0,Y 148.006,Z 616.769,A -85,B 0,C 180,E1 -23860.951,E2 -23860.951} C_VEL
LIN {X 0,Y 149.392,Z 613.791,A -85,B 0,C 180,E1 -23866.397,E2 -23866.397} C_VEL
LIN {X 0,Y 151.897,Z 609.573,A -85,B 0,C 180,E1 -23871.726,E2 -23871.726} C_VEL
LIN {X 0,Y 155.531,Z 604.004,A -85,B 0,C 180,E1 -23876.865,E2 -23876.865} C_VEL
LIN {X 0,Y 160.359,Z 596.942,A -85,B 0,C 180,E1 -23881.732,E2 -23881.732} C_VEL
LIN {X 0,Y 165.443,Z 589.402,A -85,B 0,C 180,E1 -23885.741,E2 -23885.741} C_VEL
LIN {X 0,Y 171.213,Z 580.318,A -85,B 0,C 180,E1 -23889.514,E2 -23889.514} C_VEL
LIN {X 0,Y 177.808,Z 569.417,A -85,B 0,C 180,E1 -23892.988,E2 -23892.988} C_VEL
LIN {X 0,Y 183.979,Z 558.203,A -85,B 0,C 180,E1 -23895.747,E2 -23895.747} C_VEL
LIN {X 0,Y 189.973,Z 546.021,A -85,B 0,C 180,E1 -23898.086,E2 -23898.086} C_VEL
LIN {X 0,Y 195.152,Z 533.844,A -85,B 0,C 180,E1 -23899.933,E2 -23899.933} C_VEL
LIN {X 0,Y 199.885,Z 520.911,A -85,B 0,C 180,E1 -23901.475,E2 -23901.475} C_VEL
LIN {X 0,Y 204.254,Z 506.885,A -85,B 0,C 180,E1 -23902.722,E2 -23902.722} C_VEL
LIN {X 0,Y 207.914,Z 491.858,A -85,B 0,C 180,E1 -23903.707,E2 -23903.707} C_VEL
LIN {X 0,Y 210.516,Z 476.313,A -85,B 0,C 180,E1 -23904.447,E2 -23904.447} C_VEL
LIN {X 0,Y 212.57,Z 455.538,A -85,B 0,C 180,E1 -23905.051,E2 -23905.051} C_VEL
LIN {X 0,Y 216.394,Z 406.375,A -85,B 0,C 180,E1 -23906.411,E2 -23906.411} C_VEL
LIN {X 0,Y 211.923,Z 394.863,A -85,B 0,C 180,E1 -23908.984,E2 -23908.984} C_VEL
LIN {X 0,Y 207.107,Z 384.068,A -85,B 0,C 180,E1 -23912.014,E2 -23912.014} C_VEL
LIN {X 0,Y 203.007,Z 375.792,A -85,B 0,C 180,E1 -23914.907,E2 -23914.907} C_VEL
LIN {X 0,Y 201.014,Z 372.317,A -85,B 0,C 180,E1 -23916.431,E2 -23916.431} C_VEL
LIN {X 0,Y 198.576,Z 368.622,A -85,B 0,C 180,E1 -23918.424,E2 -23918.424} C_VEL
LIN {X 0,Y 196.145,Z 365.051,A -85,B 0,C 180,E1 -23920.644,E2 -23920.644} C_VEL
LIN {X 0,Y 193.341,Z 360.937,A -85,B 0,C 180,E1 -23923.638,E2 -23923.638} C_VEL
LIN {X 0,Y 190.803,Z 357.429,A -85,B 0,C 180,E1 -23926.962,E2 -23926.962} C_VEL
LIN {X 0,Y 190.158,Z 356.313,A -85,B 0,C 180,E1 -23928.001,E2 -23928.001} C_VEL
LIN {X 0,Y 187.956,Z 353.845,A -85,B 0,C 180,E1 -23932.239,E2 -23932.239} C_VEL
LIN {X 0,Y 187.035,Z 351.164,A -85,B 0,C 180,E1 -23935.69,E2 -23935.69} C_VEL
LIN {X 0,Y 186.559,Z 350.94,A -85,B 0,C 180,E1 -23942.159,E2 -23942.159} C_VEL
LIN {X 0,Y 187.107,Z 351.384,A -85,B 0,C 180,E1 -23945.253,E2 -23945.253} C_VEL
LIN {X 0,Y 188.721,Z 355.093,A -85,B 0,C 180,E1 -23950.121,E2 -23950.121} C_VEL
LIN {X 0,Y 190.38,Z 356.601,A -85,B 0,C 180,E1 -23952.933,E2 -23952.933} C_VEL
LIN {X 0,Y 192.535,Z 360.215,A -85,B 0,C 180,E1 -23956.025,E2 -23956.025} C_VEL
LIN {X 0,Y 193.879,Z 361.747,A -85,B 0,C 180,E1 -23957.566,E2 -23957.566} C_VEL
LIN {X 0,Y 197.276,Z 366.734,A -85,B 0,C 180,E1 -23961.007,E2 -23961.007} C_VEL
LIN {X 0,Y 200.179,Z 371.041,A -85,B 0,C 180,E1 -23963.491,E2 -23963.491} C_VEL
LIN {X 0,Y 204.415,Z 377.536,A -85,B 0,C 180,E1 -23966.629,E2 -23966.629} C_VEL
LIN {X 0,Y 208.751,Z 384.893,A -85,B 0,C 180,E1 -23969.453,E2 -23969.453} C_VEL
LIN {X 0,Y 214.19,Z 394.872,A -85,B 0,C 180,E1 -23972.581,E2 -23972.581} C_VEL
LIN {X 0,Y 216.846,Z 400.265,A -85,B 0,C 180,E1 -23973.992,E2 -23973.992} C_VEL
LIN {X 0,Y 211.771,Z 462.884,A -85,B 0,C 180,E1 -23975.722,E2 -23975.722} C_VEL
LIN {X 0,Y 209.49,Z 478.175,A -85,B 0,C 180,E1 -23976.373,E2 -23976.373} C_VEL
LIN {X 0,Y 206.248,Z 493.736,A -85,B 0,C 180,E1 -23977.401,E2 -23977.401} C_VEL
LIN {X 0,Y 202.112,Z 508.637,A -85,B 0,C 180,E1 -23978.749,E2 -23978.749} C_VEL
LIN {X 0,Y 197.435,Z 522.587,A -85,B 0,C 180,E1 -23980.457,E2 -23980.457} C_VEL
LIN {X 0,Y 191.84,Z 536.014,A -85,B 0,C 180,E1 -23982.499,E2 -23982.499} C_VEL
LIN {X 0,Y 186.009,Z 548.197,A -85,B 0,C 180,E1 -23984.891,E2 -23984.891} C_VEL
LIN {X 0,Y 179.939,Z 559.297,A -85,B 0,C 180,E1 -23987.642,E2 -23987.642} C_VEL
LIN {X 0,Y 173.66,Z 570.054,A -85,B 0,C 180,E1 -23991.148,E2 -23991.148} C_VEL
LIN {X 0,Y 167.759,Z 578.992,A -85,B 0,C 180,E1 -23994.826,E2 -23994.826} C_VEL
LIN {X 0,Y 162.602,Z 586.389,A -85,B 0,C 180,E1 -23998.756,E2 -23998.756} C_VEL
LIN {X 0,Y 157.649,Z 593.293,A -85,B 0,C 180,E1 -24003.524,E2 -24003.524} C_VEL
LIN {X 0,Y 153.744,Z 598.707,A -85,B 0,C 180,E1 -24008.548,E2 -24008.548} C_VEL
LIN {X 0,Y 150.859,Z 602.785,A -85,B 0,C 180,E1 -24013.767,E2 -24013.767} C_VEL
LIN {X 0,Y 149.01,Z 605.64,A -85,B 0,C 180,E1 -24019.124,E2 -24019.124} C_VEL
LIN {X 0,Y 148.11,Z 607.347,A -85,B 0,C 180,E1 -24024.553,E2 -24024.553} C_VEL
LIN {X 0,Y 147.881,Z 607.939,A -85,B 0,C 180,E1 -24029.999,E2 -24029.999} C_VEL
LIN {X 0,Y 148.11,Z 607.381,A -85,B 0,C 180,E1 -24035.444,E2 -24035.444} C_VEL
LIN {X 0,Y 149.007,Z 605.718,A -85,B 0,C 180,E1 -24040.873,E2 -24040.873} C_VEL
LIN {X 0,Y 150.798,Z 602.905,A -85,B 0,C 180,E1 -24046.237,E2 -24046.237} C_VEL
LIN {X 0,Y 153.694,Z 598.865,A -85,B 0,C 180,E1 -24051.457,E2 -24051.457} C_VEL
LIN {X 0,Y 157.561,Z 593.502,A -85,B 0,C 180,E1 -24056.489,E2 -24056.489} C_VEL
LIN {X 0,Y 162.53,Z 586.656,A -85,B 0,C 180,E1 -24061.257,E2 -24061.257} C_VEL
LIN {X 0,Y 168.461,Z 578.101,A -85,B 0,C 180,E1 -24065.736,E2 -24065.736} C_VEL
LIN {X 0,Y 174.42,Z 568.994,A -85,B 0,C 180,E1 -24069.391,E2 -24069.391} C_VEL
LIN {X 0,Y 179.837,Z 559.725,A -85,B 0,C 180,E1 -24072.385,E2 -24072.385} C_VEL
LIN {X 0,Y 186.421,Z 547.7,A -85,B 0,C 180,E1 -24075.362,E2 -24075.362} C_VEL
LIN {X 0,Y 192.253,Z 535.417,A -85,B 0,C 180,E1 -24077.752,E2 -24077.752} C_VEL
LIN {X 0,Y 197.823,Z 521.849,A -85,B 0,C 180,E1 -24079.801,E2 -24079.801} C_VEL
LIN {X 0,Y 202.421,Z 508.119,A -85,B 0,C 180,E1 -24081.453,E2 -24081.453} C_VEL
LIN {X 0,Y 206.427,Z 493.738,A -85,B 0,C 180,E1 -24082.732,E2 -24082.732} C_VEL
LIN {X 0,Y 209.662,Z 478.466,A -85,B 0,C 180,E1 -24083.729,E2 -24083.729} C_VEL
LIN {X 0,Y 211.907,Z 463.037,A -85,B 0,C 180,E1 -24084.418,E2 -24084.418} C_VEL
LIN {X 0,Y 217.049,Z 400.579,A -85,B 0,C 180,E1 -24086.115,E2 -24086.115} C_VEL
LIN {X 0,Y 212.848,Z 392.122,A -85,B 0,C 180,E1 -24088.387,E2 -24088.387} C_VEL
LIN {X 0,Y 207.59,Z 382.723,A -85,B 0,C 180,E1 -24091.522,E2 -24091.522} C_VEL
LIN {X 0,Y 203.673,Z 376.26,A -85,B 0,C 180,E1 -24094.16,E2 -24094.16} C_VEL
LIN {X 0,Y 199.411,Z 369.664,A -85,B 0,C 180,E1 -24097.454,E2 -24097.454} C_VEL
LIN {X 0,Y 196.305,Z 365.22,A -85,B 0,C 180,E1 -24100.252,E2 -24100.252} C_VEL
LIN {X 0,Y 193.411,Z 361.018,A -85,B 0,C 180,E1 -24103.372,E2 -24103.372} C_VEL
LIN {X 0,Y 191.162,Z 358.05,A -85,B 0,C 180,E1 -24106.31,E2 -24106.31} C_VEL
LIN {X 0,Y 190.377,Z 356.479,A -85,B 0,C 180,E1 -24107.609,E2 -24107.609} C_VEL
LIN {X 0,Y 188.153,Z 354.086,A -85,B 0,C 180,E1 -24111.948,E2 -24111.948} C_VEL
LIN {X 0,Y 187.223,Z 351.29,A -85,B 0,C 180,E1 -24115.694,E2 -24115.694} C_VEL
LIN {X 0,Y 186.799,Z 350.93,A -85,B 0,C 180,E1 -24120,E2 -24120} C_VEL
LIN {X 0,Y 187.254,Z 351.463,A -85,B 0,C 180,E1 -24124.035,E2 -24124.035} C_VEL
LIN {X 0,Y 189.054,Z 355.366,A -85,B 0,C 180,E1 -24129.63,E2 -24129.63} C_VEL
LIN {X 0,Y 190.587,Z 356.778,A -85,B 0,C 180,E1 -24132.241,E2 -24132.241} C_VEL
LIN {X 0,Y 192.888,Z 360.416,A -85,B 0,C 180,E1 -24135.52,E2 -24135.52} C_VEL
LIN {X 0,Y 194.028,Z 361.814,A -85,B 0,C 180,E1 -24136.844,E2 -24136.844} C_VEL
LIN {X 0,Y 197.424,Z 366.74,A -85,B 0,C 180,E1 -24140.309,E2 -24140.309} C_VEL
LIN {X 0,Y 200.203,Z 370.926,A -85,B 0,C 180,E1 -24142.715,E2 -24142.715} C_VEL
LIN {X 0,Y 202.304,Z 374.299,A -85,B 0,C 180,E1 -24144.364,E2 -24144.364} C_VEL
LIN {X 0,Y 206.142,Z 381.838,A -85,B 0,C 180,E1 -24147.163,E2 -24147.163} C_VEL
LIN {X 0,Y 210.74,Z 391.89,A -85,B 0,C 180,E1 -24150.153,E2 -24150.153} C_VEL
LIN {X 0,Y 215.343,Z 403.139,A -85,B 0,C 180,E1 -24152.859,E2 -24152.859} C_VEL
LIN {X 0,Y 216.582,Z 406.511,A -85,B 0,C 180,E1 -24153.556,E2 -24153.556} C_VEL
LIN {X 0,Y 211.577,Z 469.23,A -85,B 0,C 180,E1 -24155.286,E2 -24155.286} C_VEL
LIN {X 0,Y 209.384,Z 484.991,A -85,B 0,C 180,E1 -24155.89,E2 -24155.89} C_VEL
LIN {X 0,Y 206.195,Z 500.323,A -85,B 0,C 180,E1 -24156.778,E2 -24156.778} C_VEL
LIN {X 0,Y 202.405,Z 513.874,A -85,B 0,C 180,E1 -24157.822,E2 -24157.822} C_VEL
LIN {X 0,Y 198.745,Z 524.871,A -85,B 0,C 180,E1 -24158.91,E2 -24158.91} C_VEL
LIN {X 0,Y 196.446,Z 530.092,A -85,B 0,C 180,E1 -24159.367,E2 -24159.367} C_VEL
LIN {X 0,Y 191.147,Z 538.358,A -85,B 0,C 180,E1 -24159.828,E2 -24159.828} C_VEL
LIN {X 0,Y 185.574,Z 546.299,A -85,B 0,C 180,E1 -24160.447,E2 -24160.447} C_VEL
LIN {X 0,Y 182.876,Z 551.005,A -85,B 0,C 180,E1 -24161.166,E2 -24161.166} C_VEL
LIN {X 0,Y 176.898,Z 562.12,A -85,B 0,C 180,E1 -24163.528,E2 -24163.528} C_VEL
LIN {X 0,Y 170.619,Z 572.651,A -85,B 0,C 180,E1 -24166.375,E2 -24166.375} C_VEL
LIN {X 0,Y 164.827,Z 581.594,A -85,B 0,C 180,E1 -24169.442,E2 -24169.442} C_VEL
LIN {X 0,Y 158.858,Z 590.416,A -85,B 0,C 180,E1 -24173.328,E2 -24173.328} C_VEL
LIN {X 0,Y 154.346,Z 596.813,A -85,B 0,C 180,E1 -24176.88,E2 -24176.88} C_VEL
LIN {X 0,Y 149.163,Z 603.838,A -85,B 0,C 180,E1 -24181.892,E2 -24181.892} C_VEL
LIN {X 0,Y 145.236,Z 609.377,A -85,B 0,C 180,E1 -24187.226,E2 -24187.226} C_VEL
LIN {X 0,Y 142.517,Z 613.578,A -85,B 0,C 180,E1 -24192.791,E2 -24192.791} C_VEL
LIN {X 0,Y 140.999,Z 616.538,A -85,B 0,C 180,E1 -24198.501,E2 -24198.501} C_VEL
LIN {X 0,Y 140.541,Z 618.317,A -85,B 0,C 180,E1 -24204.261,E2 -24204.261} C_VEL
LIN {X 0,Y 140.717,Z 618.934,A -85,B 0,C 180,E1 -24210.001,E2 -24210.001} C_VEL
LIN {X 0,Y 140.542,Z 618.299,A -85,B 0,C 180,E1 -24215.741,E2 -24215.741} C_VEL
LIN {X 0,Y 141,Z 616.496,A -85,B 0,C 180,E1 -24221.502,E2 -24221.502} C_VEL
LIN {X 0,Y 142.517,Z 613.517,A -85,B 0,C 180,E1 -24227.212,E2 -24227.212} C_VEL
LIN {X 0,Y 145.243,Z 609.298,A -85,B 0,C 180,E1 -24232.776,E2 -24232.776} C_VEL
LIN {X 0,Y 149.15,Z 603.729,A -85,B 0,C 180,E1 -24238.114,E2 -24238.114} C_VEL
LIN {X 0,Y 154.332,Z 596.669,A -85,B 0,C 180,E1 -24243.126,E2 -24243.126} C_VEL
LIN {X 0,Y 159.661,Z 589.126,A -85,B 0,C 180,E1 -24247.249,E2 -24247.249} C_VEL
LIN {X 0,Y 165.74,Z 580.043,A -85,B 0,C 180,E1 -24251.093,E2 -24251.093} C_VEL
LIN {X 0,Y 172.644,Z 569.141,A -85,B 0,C 180,E1 -24254.607,E2 -24254.607} C_VEL
LIN {X 0,Y 179.083,Z 557.928,A -85,B 0,C 180,E1 -24257.379,E2 -24257.379} C_VEL
LIN {X 0,Y 185.383,Z 545.557,A -85,B 0,C 180,E1 -24259.758,E2 -24259.758} C_VEL
LIN {X 0,Y 191.236,Z 532.135,A -85,B 0,C 180,E1 -24261.773,E2 -24261.773} C_VEL
LIN {X 0,Y 196.169,Z 518.865,A -85,B 0,C 180,E1 -24263.286,E2 -24263.286} C_VEL
LIN {X 0,Y 200.68,Z 504.347,A -85,B 0,C 180,E1 -24264.514,E2 -24264.514} C_VEL
LIN {X 0,Y 204.261,Z 489.287,A -85,B 0,C 180,E1 -24265.45,E2 -24265.45} C_VEL
LIN {X 0,Y 206.708,Z 474.192,A -85,B 0,C 180,E1 -24266.126,E2 -24266.126} C_VEL
LIN {X 0,Y 208.931,Z 450.89,A -85,B 0,C 180,E1 -24266.772,E2 -24266.772} C_VEL
LIN {X 0,Y 212.275,Z 408.971,A -85,B 0,C 180,E1 -24267.943,E2 -24267.943} C_VEL
LIN {X 0,Y 208.264,Z 398.581,A -85,B 0,C 180,E1 -24270.427,E2 -24270.427} C_VEL
LIN {X 0,Y 204.428,Z 389.543,A -85,B 0,C 180,E1 -24273.028,E2 -24273.028} C_VEL
LIN {X 0,Y 200.558,Z 381.426,A -85,B 0,C 180,E1 -24275.94,E2 -24275.94} C_VEL
LIN {X 0,Y 198.783,Z 378.193,A -85,B 0,C 180,E1 -24277.388,E2 -24277.388} C_VEL
LIN {X 0,Y 195.021,Z 372.21,A -85,B 0,C 180,E1 -24280.802,E2 -24280.802} C_VEL
LIN {X 0,Y 191.896,Z 367.639,A -85,B 0,C 180,E1 -24284.233,E2 -24284.233} C_VEL
LIN {X 0,Y 189.428,Z 363.97,A -85,B 0,C 180,E1 -24287.683,E2 -24287.683} C_VEL
LIN {X 0,Y 188.966,Z 363.17,A -85,B 0,C 180,E1 -24288.469,E2 -24288.469} C_VEL
LIN {X 0,Y 186.873,Z 360.647,A -85,B 0,C 180,E1 -24292.776,E2 -24292.776} C_VEL
LIN {X 0,Y 186.161,Z 358.303,A -85,B 0,C 180,E1 -24295.67,E2 -24295.67} C_VEL
LIN {X 0,Y 185.612,Z 357.868,A -85,B 0,C 180,E1 -24300,E2 -24300} C_VEL
LIN {X 0,Y 186.167,Z 358.462,A -85,B 0,C 180,E1 -24305.008,E2 -24305.008} C_VEL
LIN {X 0,Y 187.756,Z 362.149,A -85,B 0,C 180,E1 -24309.97,E2 -24309.97} C_VEL
LIN {X 0,Y 189.227,Z 363.66,A -85,B 0,C 180,E1 -24312.57,E2 -24312.57} C_VEL
LIN {X 0,Y 191.464,Z 367.28,A -85,B 0,C 180,E1 -24315.843,E2 -24315.843} C_VEL
LIN {X 0,Y 192.521,Z 368.652,A -85,B 0,C 180,E1 -24317.11,E2 -24317.11} C_VEL
LIN {X 0,Y 195.54,Z 373.191,A -85,B 0,C 180,E1 -24320.308,E2 -24320.308} C_VEL
LIN {X 0,Y 198.388,Z 377.598,A -85,B 0,C 180,E1 -24322.866,E2 -24322.866} C_VEL
LIN {X 0,Y 202.366,Z 383.959,A -85,B 0,C 180,E1 -24325.952,E2 -24325.952} C_VEL
LIN {X 0,Y 206.887,Z 391.962,A -85,B 0,C 180,E1 -24329.018,E2 -24329.018} C_VEL
LIN {X 0,Y 211.851,Z 401.564,A -85,B 0,C 180,E1 -24331.991,E2 -24331.991} C_VEL
LIN {X 0,Y 212.706,Z 403.365,A -85,B 0,C 180,E1 -24332.474,E2 -24332.474} C_VEL
LIN {X 0,Y 207.675,Z 463.519,A -85,B 0,C 180,E1 -24334.145,E2 -24334.145} C_VEL
LIN {X 0,Y 205.374,Z 478.457,A -85,B 0,C 180,E1 -24334.784,E2 -24334.784} C_VEL
LIN {X 0,Y 202.018,Z 494.014,A -85,B 0,C 180,E1 -24335.803,E2 -24335.803} C_VEL
LIN {X 0,Y 197.866,Z 508.569,A -85,B 0,C 180,E1 -24337.113,E2 -24337.113} C_VEL
LIN {X 0,Y 192.901,Z 522.863,A -85,B 0,C 180,E1 -24338.851,E2 -24338.851} C_VEL
LIN {X 0,Y 187.123,Z 536.288,A -85,B 0,C 180,E1 -24340.898,E2 -24340.898} C_VEL
LIN {X 0,Y 181.073,Z 548.471,A -85,B 0,C 180,E1 -24343.301,E2 -24343.301} C_VEL
LIN {X 0,Y 174.747,Z 559.571,A -85,B 0,C 180,E1 -24346.069,E2 -24346.069} C_VEL
LIN {X 0,Y 168.177,Z 570.327,A -85,B 0,C 180,E1 -24349.627,E2 -24349.627} C_VEL
LIN {X 0,Y 161.994,Z 579.265,A -85,B 0,C 180,E1 -24353.376,E2 -24353.376} C_VEL
LIN {X 0,Y 156.565,Z 586.662,A -85,B 0,C 180,E1 -24357.406,E2 -24357.406} C_VEL
LIN {X 0,Y 151.299,Z 593.566,A -85,B 0,C 180,E1 -24362.32,E2 -24362.32} C_VEL
LIN {X 0,Y 147.153,Z 598.979,A -85,B 0,C 180,E1 -24367.536,E2 -24367.536} C_VEL
LIN {X 0,Y 144.024,Z 603.058,A -85,B 0,C 180,E1 -24372.974,E2 -24372.974} C_VEL
LIN {X 0,Y 142.025,Z 605.912,A -85,B 0,C 180,E1 -24378.582,E2 -24378.582} C_VEL
LIN {X 0,Y 141.058,Z 607.617,A -85,B 0,C 180,E1 -24384.28,E2 -24384.28} C_VEL
LIN {X 0,Y 140.797,Z 608.209,A -85,B 0,C 180,E1 -24389.999,E2 -24389.999} C_VEL
LIN {X 0,Y 141.058,Z 607.65,A -85,B 0,C 180,E1 -24395.717,E2 -24395.717} C_VEL
LIN {X 0,Y 142.021,Z 605.989,A -85,B 0,C 180,E1 -24401.415,E2 -24401.415} C_VEL
LIN {X 0,Y 143.967,Z 603.176,A -85,B 0,C 180,E1 -24407.03,E2 -24407.03} C_VEL
LIN {X 0,Y 147.097,Z 599.135,A -85,B 0,C 180,E1 -24412.47,E2 -24412.47} C_VEL
LIN {X 0,Y 151.211,Z 593.773,A -85,B 0,C 180,E1 -24417.695,E2 -24417.695} C_VEL
LIN {X 0,Y 156.474,Z 586.926,A -85,B 0,C 180,E1 -24422.613,E2 -24422.613} C_VEL
LIN {X 0,Y 162.719,Z 578.371,A -85,B 0,C 180,E1 -24427.204,E2 -24427.204} C_VEL
LIN {X 0,Y 168.975,Z 569.263,A -85,B 0,C 180,E1 -24430.924,E2 -24430.924} C_VEL
LIN {X 0,Y 174.645,Z 559.993,A -85,B 0,C 180,E1 -24433.96,E2 -24433.96} C_VEL
LIN {X 0,Y 181.505,Z 547.967,A -85,B 0,C 180,E1 -24436.957,E2 -24436.957} C_VEL
LIN {X 0,Y 187.562,Z 535.683,A -85,B 0,C 180,E1 -24439.355,E2 -24439.355} C_VEL
LIN {X 0,Y 193.324,Z 522.114,A -85,B 0,C 180,E1 -24441.406,E2 -24441.406} C_VEL
LIN {X 0,Y 197.945,Z 508.788,A -85,B 0,C 180,E1 -24443.018,E2 -24443.018} C_VEL
LIN {X 0,Y 202.217,Z 494,A -85,B 0,C 180,E1 -24444.329,E2 -24444.329} C_VEL
LIN {X 0,Y 205.541,Z 478.815,A -85,B 0,C 180,E1 -24445.314,E2 -24445.314} C_VEL
LIN {X 0,Y 207.834,Z 463.645,A -85,B 0,C 180,E1 -24445.991,E2 -24445.991} C_VEL
LIN {X 0,Y 212.912,Z 403.531,A -85,B 0,C 180,E1 -24447.643,E2 -24447.643} C_VEL
LIN {X 0,Y 207.542,Z 392.93,A -85,B 0,C 180,E1 -24450.823,E2 -24450.823} C_VEL
LIN {X 0,Y 202.768,Z 384.448,A -85,B 0,C 180,E1 -24454.036,E2 -24454.036} C_VEL
LIN {X 0,Y 198.781,Z 378.103,A -85,B 0,C 180,E1 -24457.113,E2 -24457.113} C_VEL
LIN {X 0,Y 195.061,Z 372.202,A -85,B 0,C 180,E1 -24460.532,E2 -24460.532} C_VEL
LIN {X 0,Y 192.432,Z 368.288,A -85,B 0,C 180,E1 -24463.421,E2 -24463.421} C_VEL
LIN {X 0,Y 189.589,Z 364.219,A -85,B 0,C 180,E1 -24467.353,E2 -24467.353} C_VEL
LIN {X 0,Y 188.949,Z 363.173,A -85,B 0,C 180,E1 -24468.467,E2 -24468.467} C_VEL
LIN {X 0,Y 186.804,Z 360.273,A -85,B 0,C 180,E1 -24473.384,E2 -24473.384} C_VEL
LIN {X 0,Y 186.251,Z 358.271,A -85,B 0,C 180,E1 -24476.214,E2 -24476.214} C_VEL
LIN {X 0,Y 185.933,Z 357.978,A -85,B 0,C 180,E1 -24480,E2 -24480} C_VEL
LIN {X 0,Y 186.311,Z 358.392,A -85,B 0,C 180,E1 -24483.649,E2 -24483.649} C_VEL
LIN {X 0,Y 188.067,Z 362.38,A -85,B 0,C 180,E1 -24489.432,E2 -24489.432} C_VEL
LIN {X 0,Y 189.427,Z 363.754,A -85,B 0,C 180,E1 -24491.849,E2 -24491.849} C_VEL
LIN {X 0,Y 191.868,Z 367.534,A -85,B 0,C 180,E1 -24495.4,E2 -24495.4} C_VEL
LIN {X 0,Y 192.805,Z 368.947,A -85,B 0,C 180,E1 -24496.545,E2 -24496.545} C_VEL
LIN {X 0,Y 195.789,Z 373.337,A -85,B 0,C 180,E1 -24499.699,E2 -24499.699} C_VEL
LIN {X 0,Y 198.511,Z 377.628,A -85,B 0,C 180,E1 -24502.164,E2 -24502.164} C_VEL
LIN {X 0,Y 200.467,Z 380.999,A -85,B 0,C 180,E1 -24503.776,E2 -24503.776} C_VEL
LIN {X 0,Y 204.298,Z 389.063,A -85,B 0,C 180,E1 -24506.702,E2 -24506.702} C_VEL
LIN {X 0,Y 208.209,Z 398.12,A -85,B 0,C 180,E1 -24509.373,E2 -24509.373} C_VEL
LIN {X 0,Y 212.196,Z 408.392,A -85,B 0,C 180,E1 -24511.862,E2 -24511.862} C_VEL
LIN {X 0,Y 212.512,Z 409.833,A -85,B 0,C 180,E1 -24512.086,E2 -24512.086} C_VEL
LIN {X 0,Y 207.13,Z 472.991,A -85,B 0,C 180,E1 -24513.811,E2 -24513.811} C_VEL
LIN {X 0,Y 204.591,Z 488.616,A -85,B 0,C 180,E1 -24514.47,E2 -24514.47} C_VEL
LIN {X 0,Y 201.038,Z 503.853,A -85,B 0,C 180,E1 -24515.417,E2 -24515.417} C_VEL
LIN {X 0,Y 196.839,Z 517.584,A -85,B 0,C 180,E1 -24516.551,E2 -24516.551} C_VEL
LIN {X 0,Y 191.868,Z 531.044,A -85,B 0,C 180,E1 -24518.046,E2 -24518.046} C_VEL
LIN {X 0,Y 185.963,Z 544.722,A -85,B 0,C 180,E1 -24520.055,E2 -24520.055} C_VEL
LIN {X 0,Y 182.876,Z 551.005,A -85,B 0,C 180,E1 -24521.166,E2 -24521.166} C_VEL
LIN {X 0,Y 180.103,Z 555.625,A -85,B 0,C 180,E1 -24521.948,E2 -24521.948} C_VEL
LIN {X 0,Y 174.007,Z 562.914,A -85,B 0,C 180,E1 -24522.918,E2 -24522.918} C_VEL
LIN {X 0,Y 167.702,Z 569.782,A -85,B 0,C 180,E1 -24524.048,E2 -24524.048} C_VEL
LIN {X 0,Y 164.649,Z 573.75,A -85,B 0,C 180,E1 -24525.088,E2 -24525.088} C_VEL
LIN {X 0,Y 157.478,Z 584.182,A -85,B 0,C 180,E1 -24528.918,E2 -24528.918} C_VEL
LIN {X 0,Y 151.476,Z 592.398,A -85,B 0,C 180,E1 -24532.905,E2 -24532.905} C_VEL
LIN {X 0,Y 146.883,Z 598.421,A -85,B 0,C 180,E1 -24536.618,E2 -24536.618} C_VEL
LIN {X 0,Y 141.699,Z 605.065,A -85,B 0,C 180,E1 -24541.89,E2 -24541.89} C_VEL
LIN {X 0,Y 137.808,Z 610.279,A -85,B 0,C 180,E1 -24547.514,E2 -24547.514} C_VEL
LIN {X 0,Y 135.682,Z 613.306,A -85,B 0,C 180,E1 -24551.895,E2 -24551.895} C_VEL
LIN {X 0,Y 133.977,Z 616.265,A -85,B 0,C 180,E1 -24557.889,E2 -24557.889} C_VEL
LIN {X 0,Y 133.445,Z 618.045,A -85,B 0,C 180,E1 -24563.955,E2 -24563.955} C_VEL
LIN {X 0,Y 133.62,Z 618.664,A -85,B 0,C 180,E1 -24570.001,E2 -24570.001} C_VEL
LIN {X 0,Y 133.481,Z 618.495,A -85,B 0,C 180,E1 -24573.02,E2 -24573.02} C_VEL
LIN {X 0,Y 133.582,Z 617.269,A -85,B 0,C 180,E1 -24579.083,E2 -24579.083} C_VEL
LIN {X 0,Y 134.638,Z 614.881,A -85,B 0,C 180,E1 -24585.131,E2 -24585.131} C_VEL
LIN {X 0,Y 137.02,Z 611.295,A -85,B 0,C 180,E1 -24591.043,E2 -24591.043} C_VEL
LIN {X 0,Y 140.597,Z 606.416,A -85,B 0,C 180,E1 -24596.738,E2 -24596.738} C_VEL
LIN {X 0,Y 145.421,Z 600.12,A -85,B 0,C 180,E1 -24602.116,E2 -24602.116} C_VEL
LIN {X 0,Y 150.71,Z 593.337,A -85,B 0,C 180,E1 -24606.483,E2 -24606.483} C_VEL
LIN {X 0,Y 156.628,Z 585.137,A -85,B 0,C 180,E1 -24610.589,E2 -24610.589} C_VEL
LIN {X 0,Y 163.424,Z 575.32,A -85,B 0,C 180,E1 -24614.335,E2 -24614.335} C_VEL
LIN {X 0,Y 169.76,Z 565.292,A -85,B 0,C 180,E1 -24617.296,E2 -24617.296} C_VEL
LIN {X 0,Y 176.706,Z 553.4,A -85,B 0,C 180,E1 -24619.964,E2 -24619.964} C_VEL
LIN {X 0,Y 182.699,Z 541.321,A -85,B 0,C 180,E1 -24622.13,E2 -24622.13} C_VEL
LIN {X 0,Y 188.166,Z 528.728,A -85,B 0,C 180,E1 -24623.873,E2 -24623.873} C_VEL
LIN {X 0,Y 193.293,Z 514.75,A -85,B 0,C 180,E1 -24625.351,E2 -24625.351} C_VEL
LIN {X 0,Y 197.66,Z 500.354,A -85,B 0,C 180,E1 -24626.446,E2 -24626.446} C_VEL
LIN {X 0,Y 201.028,Z 485.407,A -85,B 0,C 180,E1 -24627.296,E2 -24627.296} C_VEL
LIN {X 0,Y 203.32,Z 470.27,A -85,B 0,C 180,E1 -24627.896,E2 -24627.896} C_VEL
LIN {X 0,Y 208.298,Z 412.915,A -85,B 0,C 180,E1 -24629.453,E2 -24629.453} C_VEL
LIN {X 0,Y 208.223,Z 411.464,A -85,B 0,C 180,E1 -24629.584,E2 -24629.584} C_VEL
LIN {X 0,Y 204.37,Z 401.189,A -85,B 0,C 180,E1 -24632.196,E2 -24632.196} C_VEL
LIN {X 0,Y 200.339,Z 391.643,A -85,B 0,C 180,E1 -24635.218,E2 -24635.218} C_VEL
LIN {X 0,Y 197.269,Z 385.181,A -85,B 0,C 180,E1 -24637.793,E2 -24637.793} C_VEL
LIN {X 0,Y 194.298,Z 380.365,A -85,B 0,C 180,E1 -24640.522,E2 -24640.522} C_VEL
LIN {X 0,Y 192.608,Z 377.758,A -85,B 0,C 180,E1 -24642.277,E2 -24642.277} C_VEL
LIN {X 0,Y 190.43,Z 374.286,A -85,B 0,C 180,E1 -24644.891,E2 -24644.891} C_VEL
LIN {X 0,Y 187.866,Z 370.102,A -85,B 0,C 180,E1 -24648.81,E2 -24648.81} C_VEL
LIN {X 0,Y 185.84,Z 367.525,A -85,B 0,C 180,E1 -24653.213,E2 -24653.213} C_VEL
LIN {X 0,Y 185.175,Z 365.266,A -85,B 0,C 180,E1 -24656.192,E2 -24656.192} C_VEL
LIN {X 0,Y 184.746,Z 364.916,A -85,B 0,C 180,E1 -24660,E2 -24660} C_VEL
LIN {X 0,Y 185.212,Z 365.417,A -85,B 0,C 180,E1 -24664.625,E2 -24664.625} C_VEL
LIN {X 0,Y 186.762,Z 369.158,A -85,B 0,C 180,E1 -24669.75,E2 -24669.75} C_VEL
LIN {X 0,Y 188.053,Z 370.578,A -85,B 0,C 180,E1 -24672.135,E2 -24672.135} C_VEL
LIN {X 0,Y 190.295,Z 374.216,A -85,B 0,C 180,E1 -24675.531,E2 -24675.531} C_VEL
LIN {X 0,Y 191.521,Z 376.146,A -85,B 0,C 180,E1 -24677.072,E2 -24677.072} C_VEL
LIN {X 0,Y 193.958,Z 379.844,A -85,B 0,C 180,E1 -24679.721,E2 -24679.721} C_VEL
LIN {X 0,Y 196.437,Z 383.836,A -85,B 0,C 180,E1 -24682.066,E2 -24682.066} C_VEL
LIN {X 0,Y 199.937,Z 389.666,A -85,B 0,C 180,E1 -24684.949,E2 -24684.949} C_VEL
LIN {X 0,Y 203.54,Z 396.261,A -85,B 0,C 180,E1 -24687.575,E2 -24687.575} C_VEL
LIN {X 0,Y 207.776,Z 404.641,A -85,B 0,C 180,E1 -24690.331,E2 -24690.331} C_VEL
LIN {X 0,Y 208.71,Z 406.562,A -85,B 0,C 180,E1 -24690.899,E2 -24690.899} C_VEL
LIN {X 0,Y 203.832,Z 463.388,A -85,B 0,C 180,E1 -24692.485,E2 -24692.485} C_VEL
LIN {X 0,Y 201.53,Z 478.12,A -85,B 0,C 180,E1 -24693.101,E2 -24693.101} C_VEL
LIN {X 0,Y 198.237,Z 493.009,A -85,B 0,C 180,E1 -24694.032,E2 -24694.032} C_VEL
LIN {X 0,Y 194.034,Z 507.659,A -85,B 0,C 180,E1 -24695.32,E2 -24695.32} C_VEL
LIN {X 0,Y 189.699,Z 520.019,A -85,B 0,C 180,E1 -24696.756,E2 -24696.756} C_VEL
LIN {X 0,Y 184.329,Z 532.753,A -85,B 0,C 180,E1 -24698.59,E2 -24698.59} C_VEL
LIN {X 0,Y 177.957,Z 545.585,A -85,B 0,C 180,E1 -24700.947,E2 -24700.947} C_VEL
LIN {X 0,Y 171.803,Z 556.313,A -85,B 0,C 180,E1 -24703.437,E2 -24703.437} C_VEL
LIN {X 0,Y 165.458,Z 566.531,A -85,B 0,C 180,E1 -24706.529,E2 -24706.529} C_VEL
LIN {X 0,Y 159.903,Z 574.631,A -85,B 0,C 180,E1 -24709.586,E2 -24709.586} C_VEL
LIN {X 0,Y 153.788,Z 582.861,A -85,B 0,C 180,E1 -24713.55,E2 -24713.55} C_VEL
LIN {X 0,Y 147.656,Z 590.586,A -85,B 0,C 180,E1 -24718.427,E2 -24718.427} C_VEL
LIN {X 0,Y 142.695,Z 596.72,A -85,B 0,C 180,E1 -24723.686,E2 -24723.686} C_VEL
LIN {X 0,Y 138.702,Z 601.452,A -85,B 0,C 180,E1 -24729.224,E2 -24729.224} C_VEL
LIN {X 0,Y 136.015,Z 604.903,A -85,B 0,C 180,E1 -24735.026,E2 -24735.026} C_VEL
LIN {X 0,Y 134.411,Z 607.176,A -85,B 0,C 180,E1 -24740.974,E2 -24740.974} C_VEL
LIN {X 0,Y 133.758,Z 608.327,A -85,B 0,C 180,E1 -24746.987,E2 -24746.987} C_VEL
LIN {X 0,Y 133.71,Z 608.479,A -85,B 0,C 180,E1 -24749.999,E2 -24749.999} C_VEL
LIN {X 0,Y 134.01,Z 607.92,A -85,B 0,C 180,E1 -24756.019,E2 -24756.019} C_VEL
LIN {X 0,Y 135.063,Z 606.259,A -85,B 0,C 180,E1 -24762.012,E2 -24762.012} C_VEL
LIN {X 0,Y 137.174,Z 603.446,A -85,B 0,C 180,E1 -24767.901,E2 -24767.901} C_VEL
LIN {X 0,Y 140.535,Z 599.405,A -85,B 0,C 180,E1 -24773.581,E2 -24773.581} C_VEL
LIN {X 0,Y 144.921,Z 594.044,A -85,B 0,C 180,E1 -24779.008,E2 -24779.008} C_VEL
LIN {X 0,Y 150.526,Z 587.196,A -85,B 0,C 180,E1 -24784.073,E2 -24784.073} C_VEL
LIN {X 0,Y 157.096,Z 578.64,A -85,B 0,C 180,E1 -24788.778,E2 -24788.778} C_VEL
LIN {X 0,Y 163.658,Z 569.532,A -85,B 0,C 180,E1 -24792.558,E2 -24792.558} C_VEL
LIN {X 0,Y 168.549,Z 561.878,A -85,B 0,C 180,E1 -24795.14,E2 -24795.14} C_VEL
LIN {X 0,Y 175.055,Z 551.166,A -85,B 0,C 180,E1 -24797.963,E2 -24797.963} C_VEL
LIN {X 0,Y 181.248,Z 539.471,A -85,B 0,C 180,E1 -24800.412,E2 -24800.412} C_VEL
LIN {X 0,Y 187.164,Z 526.736,A -85,B 0,C 180,E1 -24802.473,E2 -24802.473} C_VEL
LIN {X 0,Y 192.529,Z 512.581,A -85,B 0,C 180,E1 -24804.309,E2 -24804.309} C_VEL
LIN {X 0,Y 197.22,Z 497.672,A -85,B 0,C 180,E1 -24805.719,E2 -24805.719} C_VEL
LIN {X 0,Y 200.865,Z 482.604,A -85,B 0,C 180,E1 -24806.766,E2 -24806.766} C_VEL
LIN {X 0,Y 203.424,Z 467.718,A -85,B 0,C 180,E1 -24807.494,E2 -24807.494} C_VEL
LIN {X 0,Y 205.058,Z 453.008,A -85,B 0,C 180,E1 -24807.947,E2 -24807.947} C_VEL
LIN {X 0,Y 208.9,Z 406.689,A -85,B 0,C 180,E1 -24809.231,E2 -24809.231} C_VEL
LIN {X 0,Y 204.453,Z 397.773,A -85,B 0,C 180,E1 -24812.069,E2 -24812.069} C_VEL
LIN {X 0,Y 199.954,Z 389.454,A -85,B 0,C 180,E1 -24815.336,E2 -24815.336} C_VEL
LIN {X 0,Y 195.574,Z 382.189,A -85,B 0,C 180,E1 -24819.063,E2 -24819.063} C_VEL
LIN {X 0,Y 192.935,Z 378.115,A -85,B 0,C 180,E1 -24821.723,E2 -24821.723} C_VEL
LIN {X 0,Y 190.628,Z 374.47,A -85,B 0,C 180,E1 -24824.495,E2 -24824.495} C_VEL
LIN {X 0,Y 188.361,Z 370.996,A -85,B 0,C 180,E1 -24827.885,E2 -24827.885} C_VEL
LIN {X 0,Y 187.784,Z 370.05,A -85,B 0,C 180,E1 -24828.941,E2 -24828.941} C_VEL
LIN {X 0,Y 185.816,Z 367.175,A -85,B 0,C 180,E1 -24833.768,E2 -24833.768} C_VEL
LIN {X 0,Y 185.384,Z 365.351,A -85,B 0,C 180,E1 -24836.196,E2 -24836.196} C_VEL
LIN {X 0,Y 185.068,Z 365.026,A -85,B 0,C 180,E1 -24840,E2 -24840} C_VEL
LIN {X 0,Y 185.402,Z 365.573,A -85,B 0,C 180,E1 -24843.531,E2 -24843.531} C_VEL
LIN {X 0,Y 187.206,Z 369.493,A -85,B 0,C 180,E1 -24849.475,E2 -24849.475} C_VEL
LIN {X 0,Y 188.253,Z 370.66,A -85,B 0,C 180,E1 -24851.405,E2 -24851.405} C_VEL
LIN {X 0,Y 190.591,Z 374.361,A -85,B 0,C 180,E1 -24854.958,E2 -24854.958} C_VEL
LIN {X 0,Y 194.115,Z 379.833,A -85,B 0,C 180,E1 -24859.017,E2 -24859.017} C_VEL
LIN {X 0,Y 197.628,Z 385.543,A -85,B 0,C 180,E1 -24862.283,E2 -24862.283} C_VEL
LIN {X 0,Y 201.124,Z 393.179,A -85,B 0,C 180,E1 -24865.203,E2 -24865.203} C_VEL
LIN {X 0,Y 204.812,Z 401.994,A -85,B 0,C 180,E1 -24867.939,E2 -24867.939} C_VEL
LIN {X 0,Y 208.6,Z 412.078,A -85,B 0,C 180,E1 -24870.495,E2 -24870.495} C_VEL
LIN {X 0,Y 203.223,Z 473.027,A -85,B 0,C 180,E1 -24872.159,E2 -24872.159} C_VEL
LIN {X 0,Y 200.661,Z 488.355,A -85,B 0,C 180,E1 -24872.8,E2 -24872.8} C_VEL
LIN {X 0,Y 197.014,Z 503.59,A -85,B 0,C 180,E1 -24873.736,E2 -24873.736} C_VEL
LIN {X 0,Y 192.699,Z 517.32,A -85,B 0,C 180,E1 -24874.856,E2 -24874.856} C_VEL
LIN {X 0,Y 187.57,Z 530.778,A -85,B 0,C 180,E1 -24876.336,E2 -24876.336} C_VEL
LIN {X 0,Y 181.613,Z 544.049,A -85,B 0,C 180,E1 -24878.255,E2 -24878.255} C_VEL
LIN {X 0,Y 174.928,Z 556.918,A -85,B 0,C 180,E1 -24880.684,E2 -24880.684} C_VEL
LIN {X 0,Y 167.642,Z 569.105,A -85,B 0,C 180,E1 -24883.685,E2 -24883.685} C_VEL
LIN {X 0,Y 164.649,Z 573.75,A -85,B 0,C 180,E1 -24885.088,E2 -24885.088} C_VEL
LIN {X 0,Y 161.596,Z 577.659,A -85,B 0,C 180,E1 -24886.218,E2 -24886.218} C_VEL
LIN {X 0,Y 155.132,Z 583.666,A -85,B 0,C 180,E1 -24887.863,E2 -24887.863} C_VEL
LIN {X 0,Y 148.65,Z 589.191,A -85,B 0,C 180,E1 -24889.776,E2 -24889.776} C_VEL
LIN {X 0,Y 145.645,Z 592.343,A -85,B 0,C 180,E1 -24891.327,E2 -24891.327} C_VEL
LIN {X 0,Y 139.42,Z 599.978,A -85,B 0,C 180,E1 -24896.325,E2 -24896.325} C_VEL
LIN {X 0,Y 134.234,Z 606.238,A -85,B 0,C 180,E1 -24901.889,E2 -24901.889} C_VEL
LIN {X 0,Y 130.353,Z 611.094,A -85,B 0,C 180,E1 -24907.828,E2 -24907.828} C_VEL
LIN {X 0,Y 127.729,Z 614.662,A -85,B 0,C 180,E1 -24914.033,E2 -24914.033} C_VEL
LIN {X 0,Y 126.537,Z 617.029,A -85,B 0,C 180,E1 -24920.41,E2 -24920.41} C_VEL
LIN {X 0,Y 126.381,Z 618.23,A -85,B 0,C 180,E1 -24926.814,E2 -24926.814} C_VEL
LIN {X 0,Y 126.505,Z 618.38,A -85,B 0,C 180,E1 -24930.323,E2 -24930.323} C_VEL
LIN {X 0,Y 126.357,Z 617.755,A -85,B 0,C 180,E1 -24936.388,E2 -24936.388} C_VEL
LIN {X 0,Y 126.98,Z 615.949,A -85,B 0,C 180,E1 -24942.792,E2 -24942.792} C_VEL
LIN {X 0,Y 128.892,Z 612.969,A -85,B 0,C 180,E1 -24949.098,E2 -24949.098} C_VEL
LIN {X 0,Y 132.306,Z 608.53,A -85,B 0,C 180,E1 -24955.442,E2 -24955.442} C_VEL
LIN {X 0,Y 136.652,Z 603.18,A -85,B 0,C 180,E1 -24960.952,E2 -24960.952} C_VEL
LIN {X 0,Y 142.527,Z 596.119,A -85,B 0,C 180,E1 -24966.281,E2 -24966.281} C_VEL
LIN {X 0,Y 149.353,Z 587.342,A -85,B 0,C 180,E1 -24971.209,E2 -24971.209} C_VEL
LIN {X 0,Y 156.28,Z 578.037,A -85,B 0,C 180,E1 -24975.098,E2 -24975.098} C_VEL
LIN {X 0,Y 162.755,Z 568.59,A -85,B 0,C 180,E1 -24978.151,E2 -24978.151} C_VEL
LIN {X 0,Y 169.76,Z 557.38,A -85,B 0,C 180,E1 -24980.92,E2 -24980.92} C_VEL
LIN {X 0,Y 176.394,Z 545.213,A -85,B 0,C 180,E1 -24983.259,E2 -24983.259} C_VEL
LIN {X 0,Y 182.78,Z 531.585,A -85,B 0,C 180,E1 -24985.276,E2 -24985.276} C_VEL
LIN {X 0,Y 188.014,Z 518.312,A -85,B 0,C 180,E1 -24986.762,E2 -24986.762} C_VEL
LIN {X 0,Y 192.792,Z 503.793,A -85,B 0,C 180,E1 -24987.948,E2 -24987.948} C_VEL
LIN {X 0,Y 196.558,Z 488.727,A -85,B 0,C 180,E1 -24988.861,E2 -24988.861} C_VEL
LIN {X 0,Y 199.175,Z 473.419,A -85,B 0,C 180,E1 -24989.527,E2 -24989.527} C_VEL
LIN {X 0,Y 201.664,Z 448.359,A -85,B 0,C 180,E1 -24990.207,E2 -24990.207} C_VEL
LIN {X 0,Y 204.586,Z 414.722,A -85,B 0,C 180,E1 -24991.114,E2 -24991.114} C_VEL
LIN {X 0,Y 200.803,Z 404.346,A -85,B 0,C 180,E1 -24993.917,E2 -24993.917} C_VEL
LIN {X 0,Y 197.386,Z 396.063,A -85,B 0,C 180,E1 -24996.721,E2 -24996.721} C_VEL
LIN {X 0,Y 195.08,Z 391.038,A -85,B 0,C 180,E1 -24998.815,E2 -24998.815} C_VEL
LIN {X 0,Y 191.735,Z 385.224,A -85,B 0,C 180,E1 -25002.193,E2 -25002.193} C_VEL
LIN {X 0,Y 188.866,Z 380.756,A -85,B 0,C 180,E1 -25005.728,E2 -25005.728} C_VEL
LIN {X 0,Y 186.618,Z 376.917,A -85,B 0,C 180,E1 -25009.421,E2 -25009.421} C_VEL
LIN {X 0,Y 184.587,Z 373.761,A -85,B 0,C 180,E1 -25014.538,E2 -25014.538} C_VEL
LIN {X 0,Y 184.204,Z 372.229,A -85,B 0,C 180,E1 -25016.719,E2 -25016.719} C_VEL
LIN {X 0,Y 183.965,Z 372.086,A -85,B 0,C 180,E1 -25022.19,E2 -25022.19} C_VEL
LIN {X 0,Y 184.301,Z 372.593,A -85,B 0,C 180,E1 -25024.511,E2 -25024.511} C_VEL
LIN {X 0,Y 185.774,Z 376.147,A -85,B 0,C 180,E1 -25029.527,E2 -25029.527} C_VEL
LIN {X 0,Y 186.922,Z 377.555,A -85,B 0,C 180,E1 -25031.756,E2 -25031.756} C_VEL
LIN {X 0,Y 189.031,Z 381.044,A -85,B 0,C 180,E1 -25035.085,E2 -25035.085} C_VEL
LIN {X 0,Y 192.278,Z 386.29,A -85,B 0,C 180,E1 -25038.998,E2 -25038.998} C_VEL
LIN {X 0,Y 195.882,Z 392.333,A -85,B 0,C 180,E1 -25042.478,E2 -25042.478} C_VEL
LIN {X 0,Y 200.076,Z 400.037,A -85,B 0,C 180,E1 -25045.893,E2 -25045.893} C_VEL
LIN {X 0,Y 204.697,Z 409.472,A -85,B 0,C 180,E1 -25049.151,E2 -25049.151} C_VEL
LIN {X 0,Y 204.909,Z 409.952,A -85,B 0,C 180,E1 -25049.293,E2 -25049.293} C_VEL
LIN {X 0,Y 200.031,Z 464.436,A -85,B 0,C 180,E1 -25050.801,E2 -25050.801} C_VEL
LIN {X 0,Y 197.473,Z 479.88,A -85,B 0,C 180,E1 -25051.454,E2 -25051.454} C_VEL
LIN {X 0,Y 193.748,Z 495.722,A -85,B 0,C 180,E1 -25052.5,E2 -25052.5} C_VEL
LIN {X 0,Y 189.331,Z 509.977,A -85,B 0,C 180,E1 -25053.778,E2 -25053.778} C_VEL
LIN {X 0,Y 184.335,Z 523.412,A -85,B 0,C 180,E1 -25055.415,E2 -25055.415} C_VEL
LIN {X 0,Y 178.156,Z 536.837,A -85,B 0,C 180,E1 -25057.446,E2 -25057.446} C_VEL
LIN {X 0,Y 171.657,Z 549.017,A -85,B 0,C 180,E1 -25059.853,E2 -25059.853} C_VEL
LIN {X 0,Y 164.788,Z 560.119,A -85,B 0,C 180,E1 -25062.632,E2 -25062.632} C_VEL
LIN {X 0,Y 157.595,Z 570.874,A -85,B 0,C 180,E1 -25066.271,E2 -25066.271} C_VEL
LIN {X 0,Y 150.806,Z 579.811,A -85,B 0,C 180,E1 -25070.147,E2 -25070.147} C_VEL
LIN {X 0,Y 144.762,Z 587.208,A -85,B 0,C 180,E1 -25074.366,E2 -25074.366} C_VEL
LIN {X 0,Y 138.838,Z 594.112,A -85,B 0,C 180,E1 -25079.587,E2 -25079.587} C_VEL
LIN {X 0,Y 134.106,Z 599.523,A -85,B 0,C 180,E1 -25085.211,E2 -25085.211} C_VEL
LIN {X 0,Y 130.472,Z 603.602,A -85,B 0,C 180,E1 -25091.142,E2 -25091.142} C_VEL
LIN {X 0,Y 128.112,Z 606.455,A -85,B 0,C 180,E1 -25097.323,E2 -25097.323} C_VEL
LIN {X 0,Y 126.956,Z 608.158,A -85,B 0,C 180,E1 -25103.642,E2 -25103.642} C_VEL
LIN {X 0,Y 126.633,Z 608.749,A -85,B 0,C 180,E1 -25109.998,E2 -25109.998} C_VEL
LIN {X 0,Y 126.956,Z 608.19,A -85,B 0,C 180,E1 -25116.355,E2 -25116.355} C_VEL
LIN {X 0,Y 128.105,Z 606.53,A -85,B 0,C 180,E1 -25122.675,E2 -25122.675} C_VEL
LIN {X 0,Y 130.423,Z 603.717,A -85,B 0,C 180,E1 -25128.862,E2 -25128.862} C_VEL
LIN {X 0,Y 134.022,Z 599.676,A -85,B 0,C 180,E1 -25134.802,E2 -25134.802} C_VEL
LIN {X 0,Y 138.975,Z 593.993,A -85,B 0,C 180,E1 -25140.717,E2 -25140.717} C_VEL
LIN {X 0,Y 144.67,Z 587.466,A -85,B 0,C 180,E1 -25145.657,E2 -25145.657} C_VEL
LIN {X 0,Y 151.598,Z 578.91,A -85,B 0,C 180,E1 -25150.467,E2 -25150.467} C_VEL
LIN {X 0,Y 158.469,Z 569.802,A -85,B 0,C 180,E1 -25154.305,E2 -25154.305} C_VEL
LIN {X 0,Y 164.707,Z 560.53,A -85,B 0,C 180,E1 -25157.395,E2 -25157.395} C_VEL
LIN {X 0,Y 172.125,Z 548.501,A -85,B 0,C 180,E1 -25160.414,E2 -25160.414} C_VEL
LIN {X 0,Y 178.658,Z 536.215,A -85,B 0,C 180,E1 -25162.804,E2 -25162.804} C_VEL
LIN {X 0,Y 184.613,Z 523.129,A -85,B 0,C 180,E1 -25164.782,E2 -25164.782} C_VEL
LIN {X 0,Y 189.513,Z 510.023,A -85,B 0,C 180,E1 -25166.36,E2 -25166.36} C_VEL
LIN {X 0,Y 193.966,Z 495.681,A -85,B 0,C 180,E1 -25167.637,E2 -25167.637} C_VEL
LIN {X 0,Y 197.673,Z 480.068,A -85,B 0,C 180,E1 -25168.652,E2 -25168.652} C_VEL
LIN {X 0,Y 200.093,Z 465.24,A -85,B 0,C 180,E1 -25169.318,E2 -25169.318} C_VEL
LIN {X 0,Y 203.985,Z 423.421,A -85,B 0,C 180,E1 -25170.459,E2 -25170.459} C_VEL
LIN {X 0,Y 205.061,Z 409.94,A -85,B 0,C 180,E1 -25170.871,E2 -25170.871} C_VEL
LIN {X 0,Y 200.567,Z 400.764,A -85,B 0,C 180,E1 -25174.023,E2 -25174.023} C_VEL
LIN {X 0,Y 196.971,Z 394.113,A -85,B 0,C 180,E1 -25176.891,E2 -25176.891} C_VEL
LIN {X 0,Y 193.445,Z 388.067,A -85,B 0,C 180,E1 -25180.155,E2 -25180.155} C_VEL
LIN {X 0,Y 191.292,Z 384.598,A -85,B 0,C 180,E1 -25182.48,E2 -25182.48} C_VEL
LIN {X 0,Y 189.165,Z 381.08,A -85,B 0,C 180,E1 -25185.201,E2 -25185.201} C_VEL
LIN {X 0,Y 186.918,Z 377.231,A -85,B 0,C 180,E1 -25188.89,E2 -25188.89} C_VEL
LIN {X 0,Y 184.714,Z 373.748,A -85,B 0,C 180,E1 -25194.701,E2 -25194.701} C_VEL
LIN {X 0,Y 184.431,Z 372.304,A -85,B 0,C 180,E1 -25196.723,E2 -25196.723} C_VEL
LIN {X 0,Y 184.35,Z 372.211,A -85,B 0,C 180,E1 -25202.185,E2 -25202.185} C_VEL
LIN {X 0,Y 184.52,Z 372.766,A -85,B 0,C 180,E1 -25203.548,E2 -25203.548} C_VEL
LIN {X 0,Y 186.201,Z 376.476,A -85,B 0,C 180,E1 -25209.231,E2 -25209.231} C_VEL
LIN {X 0,Y 187.1,Z 377.523,A -85,B 0,C 180,E1 -25210.962,E2 -25210.962} C_VEL
LIN {X 0,Y 189.798,Z 382.03,A -85,B 0,C 180,E1 -25215.16,E2 -25215.16} C_VEL
LIN {X 0,Y 192.441,Z 386.306,A -85,B 0,C 180,E1 -25218.295,E2 -25218.295} C_VEL
LIN {X 0,Y 195.522,Z 391.547,A -85,B 0,C 180,E1 -25221.34,E2 -25221.34} C_VEL
LIN {X 0,Y 198.593,Z 398.505,A -85,B 0,C 180,E1 -25224.084,E2 -25224.084} C_VEL
LIN {X 0,Y 202.166,Z 407.628,A -85,B 0,C 180,E1 -25226.939,E2 -25226.939} C_VEL
LIN {X 0,Y 204.794,Z 414.89,A -85,B 0,C 180,E1 -25228.854,E2 -25228.854} C_VEL
LIN {X 0,Y 199.593,Z 472.394,A -85,B 0,C 180,E1 -25230.421,E2 -25230.421} C_VEL
LIN {X 0,Y 196.899,Z 488.094,A -85,B 0,C 180,E1 -25231.06,E2 -25231.06} C_VEL
LIN {X 0,Y 193.163,Z 503.326,A -85,B 0,C 180,E1 -25231.986,E2 -25231.986} C_VEL
LIN {X 0,Y 188.727,Z 517.055,A -85,B 0,C 180,E1 -25233.085,E2 -25233.085} C_VEL
LIN {X 0,Y 183.433,Z 530.511,A -85,B 0,C 180,E1 -25234.54,E2 -25234.54} C_VEL
LIN {X 0,Y 177.549,Z 543.226,A -85,B 0,C 180,E1 -25236.355,E2 -25236.355} C_VEL
LIN {X 0,Y 170.972,Z 555.577,A -85,B 0,C 180,E1 -25238.648,E2 -25238.648} C_VEL
LIN {X 0,Y 163.904,Z 567.071,A -85,B 0,C 180,E1 -25241.379,E2 -25241.379} C_VEL
LIN {X 0,Y 157.322,Z 576.755,A -85,B 0,C 180,E1 -25244.378,E2 -25244.378} C_VEL
LIN {X 0,Y 150.326,Z 586.281,A -85,B 0,C 180,E1 -25248.226,E2 -25248.226} C_VEL
LIN {X 0,Y 145.645,Z 592.343,A -85,B 0,C 180,E1 -25251.327,E2 -25251.327} C_VEL
LIN {X 0,Y 142.702,Z 595.344,A -85,B 0,C 180,E1 -25252.979,E2 -25252.979} C_VEL
LIN {X 0,Y 136.446,Z 599.905,A -85,B 0,C 180,E1 -25255.528,E2 -25255.528} C_VEL
LIN {X 0,Y 130.361,Z 603.949,A -85,B 0,C 180,E1 -25258.414,E2 -25258.414} C_VEL
LIN {X 0,Y 127.784,Z 606.137,A -85,B 0,C 180,E1 -25260.565,E2 -25260.565} C_VEL
LIN {X 0,Y 123.742,Z 610.821,A -85,B 0,C 180,E1 -25266.575,E2 -25266.575} C_VEL
LIN {X 0,Y 120.851,Z 614.39,A -85,B 0,C 180,E1 -25273.098,E2 -25273.098} C_VEL
LIN {X 0,Y 119.482,Z 616.756,A -85,B 0,C 180,E1 -25279.838,E2 -25279.838} C_VEL
LIN {X 0,Y 119.28,Z 617.96,A -85,B 0,C 180,E1 -25286.624,E2 -25286.624} C_VEL
LIN {X 0,Y 119.438,Z 618.123,A -85,B 0,C 180,E1 -25290.002,E2 -25290.002} C_VEL
LIN {X 0,Y 119.281,Z 617.953,A -85,B 0,C 180,E1 -25293.379,E2 -25293.379} C_VEL
LIN {X 0,Y 119.482,Z 616.724,A -85,B 0,C 180,E1 -25300.165,E2 -25300.165} C_VEL
LIN {X 0,Y 120.851,Z 614.334,A -85,B 0,C 180,E1 -25306.906,E2 -25306.906} C_VEL
LIN {X 0,Y 123.747,Z 610.747,A -85,B 0,C 180,E1 -25313.427,E2 -25313.427} C_VEL
LIN {X 0,Y 127.928,Z 605.866,A -85,B 0,C 180,E1 -25319.634,E2 -25319.634} C_VEL
LIN {X 0,Y 133.479,Z 599.57,A -85,B 0,C 180,E1 -25325.394,E2 -25325.394} C_VEL
LIN {X 0,Y 140.302,Z 591.687,A -85,B 0,C 180,E1 -25330.634,E2 -25330.634} C_VEL
LIN {X 0,Y 146.054,Z 584.585,A -85,B 0,C 180,E1 -25334.247,E2 -25334.247} C_VEL
LIN {X 0,Y 153.533,Z 574.771,A -85,B 0,C 180,E1 -25338.062,E2 -25338.062} C_VEL
LIN {X 0,Y 160.436,Z 564.743,A -85,B 0,C 180,E1 -25341.039,E2 -25341.039} C_VEL
LIN {X 0,Y 167.793,Z 552.978,A -85,B 0,C 180,E1 -25343.675,E2 -25343.675} C_VEL
LIN {X 0,Y 174.643,Z 540.077,A -85,B 0,C 180,E1 -25345.946,E2 -25345.946} C_VEL
LIN {X 0,Y 180.824,Z 526.589,A -85,B 0,C 180,E1 -25347.711,E2 -25347.711} C_VEL
LIN {X 0,Y 186.285,Z 512.207,A -85,B 0,C 180,E1 -25349.128,E2 -25349.128} C_VEL
LIN {X 0,Y 190.866,Z 497.192,A -85,B 0,C 180,E1 -25350.184,E2 -25350.184} C_VEL
LIN {X 0,Y 194.206,Z 482.29,A -85,B 0,C 180,E1 -25350.949,E2 -25350.949} C_VEL
LIN {X 0,Y 196.377,Z 467.766,A -85,B 0,C 180,E1 -25351.458,E2 -25351.458} C_VEL
LIN {X 0,Y 200.944,Z 417.55,A -85,B 0,C 180,E1 -25352.816,E2 -25352.816} C_VEL
LIN {X 0,Y 197.274,Z 407.22,A -85,B 0,C 180,E1 -25355.817,E2 -25355.817} C_VEL
LIN {X 0,Y 194.193,Z 399.497,A -85,B 0,C 180,E1 -25358.644,E2 -25358.644} C_VEL
LIN {X 0,Y 191.951,Z 394.898,A -85,B 0,C 180,E1 -25360.899,E2 -25360.899} C_VEL
LIN {X 0,Y 189.347,Z 390.575,A -85,B 0,C 180,E1 -25363.837,E2 -25363.837} C_VEL
LIN {X 0,Y 187.572,Z 387.522,A -85,B 0,C 180,E1 -25366.25,E2 -25366.25} C_VEL
LIN {X 0,Y 185.464,Z 383.793,A -85,B 0,C 180,E1 -25369.906,E2 -25369.906} C_VEL
LIN {X 0,Y 183.585,Z 380.587,A -85,B 0,C 180,E1 -25375.059,E2 -25375.059} C_VEL
LIN {X 0,Y 183.337,Z 379.302,A -85,B 0,C 180,E1 -25376.704,E2 -25376.704} C_VEL
LIN {X 0,Y 183.099,Z 379.138,A -85,B 0,C 180,E1 -25382.2,E2 -25382.2} C_VEL
LIN {X 0,Y 183.378,Z 379.624,A -85,B 0,C 180,E1 -25384.259,E2 -25384.259} C_VEL
LIN {X 0,Y 184.786,Z 383.149,A -85,B 0,C 180,E1 -25389.302,E2 -25389.302} C_VEL
LIN {X 0,Y 185.711,Z 384.311,A -85,B 0,C 180,E1 -25391.187,E2 -25391.187} C_VEL
LIN {X 0,Y 188.331,Z 388.867,A -85,B 0,C 180,E1 -25395.42,E2 -25395.42} C_VEL
LIN {X 0,Y 191.023,Z 393.483,A -85,B 0,C 180,E1 -25398.711,E2 -25398.711} C_VEL
LIN {X 0,Y 194.12,Z 398.95,A -85,B 0,C 180,E1 -25401.829,E2 -25401.829} C_VEL
LIN {X 0,Y 197.915,Z 406.194,A -85,B 0,C 180,E1 -25405.082,E2 -25405.082} C_VEL
LIN {X 0,Y 201.255,Z 413.325,A -85,B 0,C 180,E1 -25407.615,E2 -25407.615} C_VEL
LIN {X 0,Y 196.492,Z 464.821,A -85,B 0,C 180,E1 -25409.034,E2 -25409.034} C_VEL
LIN {X 0,Y 194.046,Z 479.301,A -85,B 0,C 180,E1 -25409.628,E2 -25409.628} C_VEL
LIN {X 0,Y 190.361,Z 494.848,A -85,B 0,C 180,E1 -25410.604,E2 -25410.604} C_VEL
LIN {X 0,Y 185.803,Z 509.41,A -85,B 0,C 180,E1 -25411.876,E2 -25411.876} C_VEL
LIN {X 0,Y 180.319,Z 523.687,A -85,B 0,C 180,E1 -25413.58,E2 -25413.58} C_VEL
LIN {X 0,Y 173.933,Z 537.111,A -85,B 0,C 180,E1 -25415.59,E2 -25415.59} C_VEL
LIN {X 0,Y 167.182,Z 549.292,A -85,B 0,C 180,E1 -25417.979,E2 -25417.979} C_VEL
LIN {X 0,Y 160.048,Z 560.393,A -85,B 0,C 180,E1 -25420.756,E2 -25420.756} C_VEL
